ELSIF SpeedUpSubState=SpeedUpCS AND gait_cycle-EnterSpeedUpCSCount=LREAL_TO_UDINT(Time_CS*gvl.sampleRate) THEN
	SpeedUpSubState:=SpeedUpDS;
	EnterSpeedUpDSCount:=gait_cycle;
	body_ref_pos_enter :=body_ref_pos;
	body_ref_ang_enter:=body_ref_ang;
	leg_ref_pos_enter := leg_ref_pos;
ELSIF SpeedUpSubState=SpeedUpDS AND gait_cycle-EnterSpeedUpDSCount=LREAL_TO_UDINT(Time_DS*gvl.sampleRate) THEN
	SpeedUpSubState:=SpeedUpSS;
	EnterSpeedUpSPCount:=gait_cycle;
	body_ref_pos_enter :=body_ref_pos;
	body_ref_ang_enter:=body_ref_ang;
	leg_ref_pos_enter := leg_ref_pos;
	SpeedUpFinished:=TRUE;
	tipForceDesire:=tipForceDesireZeros;
	RequireSlide:=TRUE;
END_IF

body_ref_pos:=body_ref_pos_enter;
body_ref_ang:=body_ref_ang_enter;
leg_ref_pos:=leg_ref_pos_enter;

IF SpeedUpSubState=SpeedUpAS AND gait_cycle-EnterSpeedUpASCount<=Time_AS*gvl.sampleRate THEN
	fbHermitInterpolation(t0:=EnterSpeedUpASCount*delta_t , T:=Time_AS , y0:=0 , 
		y1:=Distance_x_AS , v0:=0 , v1:=target_vel , tNow:=gait_cycle* delta_t, 
		y=> body_ref_pos_wrt_body.data[0], v=>invalid );	
	body_ref_pos_wrt_body.data[1]:=0;body_ref_pos_wrt_body.data[2]:=0;
	fbRotMat(yaw := body_ref_ang_enter.data[2], pitch := body_ref_ang_enter.data[1],roll := body_ref_ang_enter.data[0], rm =>  Rb_target1 );
	body_ref_pos:=VecAdd(body_ref_pos_enter,MatMulVec(Rb_target1,body_ref_pos_wrt_body));
	
	//force compensator
	tipForceTarget:=tipForceDesireLegAF;
	IF (gait_cycle-EnterSpeedUpASCount)<=fceLoadTime*gvl.sampleRate THEN
		tr  := UDINT_TO_LREAL(gait_cycle-EnterSpeedUpASCount) / gvl.sampleRate / fceLoadTime;
		fbGetPivot(tNow := tr, tTotal := 1.0, pivot => pvt);
		FOR i:=0 TO 5 DO
			FOR j:=0 TO 2 DO
				tipForceDesire[i,j]:=(1-pvt)*tipForceDesireZeros[i,j]+pvt*tipForceTarget[i,j];
			END_FOR
		END_FOR	
	END_IF
	
END_IF
	//force compensator
	tipForceTarget:=tipForceDesireLegAF;
	IF (gait_cycle-EnterSpeedUpASCount)>(Time_AS+Time_CS-fceLoadTime)*gvl.sampleRate AND (gait_cycle-EnterSpeedUpASCount)<=(Time_AS+Time_CS)*gvl.sampleRate THEN
		tr  := (UDINT_TO_LREAL(gait_cycle-EnterSpeedUpASCount) / gvl.sampleRate- (Time_AS+Time_CS-fceLoadTime))/ fceLoadTime;
		fbGetPivot(tNow := tr, tTotal := 1.0, pivot => pvt);
		FOR i:=0 TO 5 DO
			FOR j:=0 TO 2 DO
				tipForceDesire[i,j]:=(1-pvt)*tipForceTarget[i,j]+pvt*tipForceDesireZeros[i,j];
			END_FOR
		END_FOR	
	END_IF

IF SpeedUpSubState=SpeedUpCS AND gait_cycle-EnterSpeedUpCSCount<=Time_CS*gvl.sampleRate THEN
	fbHermitInterpolation(t0:=EnterSpeedUpCSCount*delta_t , T:=Time_CS , y0:=0 , 
		y1:=target_vel*Time_CS , v0:=target_vel , v1:=target_vel , tNow:=gait_cycle* delta_t, 
		y=> body_ref_pos_wrt_body.data[0], v=>invalid );
	body_ref_pos_wrt_body.data[1]:=0;body_ref_pos_wrt_body.data[2]:=0;
	fbRotMat(yaw := body_ref_ang_enter.data[2], pitch := body_ref_ang_enter.data[1],roll := body_ref_ang_enter.data[0], rm =>  Rb_target1 );
	body_ref_pos:=VecAdd(body_ref_pos_enter,MatMulVec(Rb_target1,body_ref_pos_wrt_body));
END_IF
IF SpeedUpSubState=SpeedUpDS AND gait_cycle-EnterSpeedUpDSCount<=Time_DS*gvl.sampleRate THEN
	fbHermitInterpolation(t0:=EnterSpeedUpDSCount*delta_t , T:=Time_DS , y0:=0 , 
		y1:=Distance_x_DS , v0:=target_vel , v1:=0 , tNow:=gait_cycle* delta_t, 
		y=> body_ref_pos_wrt_body.data[0], v=>invalid );
	body_ref_pos_wrt_body.data[1]:=0;body_ref_pos_wrt_body.data[2]:=0;
	
	fbRotMat(yaw := body_ref_ang_enter.data[2], pitch := body_ref_ang_enter.data[1],roll := body_ref_ang_enter.data[0], rm =>  Rb_target1 );
	body_ref_pos:=VecAdd(body_ref_pos_enter,MatMulVec(Rb_target1,body_ref_pos_wrt_body));
	
	tr  := UDINT_TO_LREAL(gait_cycle - EnterSpeedUpDSCount) / gvl.sampleRate / Time_DS;
	fbGetPivot(tNow := tr, tTotal := 1.0, pivot => pvt);
	FOR i:=0 TO 1 DO
		leg_ref_pos[Mapping05[i]].data[2]:=(1-pvt)*leg_ref_pos_enter[Mapping05[i]].data[2]+pvt*(leg_ref_pos_enter[Mapping05[i]].data[2]+Distance_y_DS);
	END_FOR
	
END_IF
IF SpeedUpSubState=SpeedUpAS OR SpeedUpSubState=SpeedUpCS OR SpeedUpSubState=SpeedUpDS THEN
	FOR i:=0 TO 1 DO
		gvl.legCtrl[Mapping14[i]].ForwardKinetics(motorAngles:=SpeedUp_MJntRef[i].data , legIndex:=Mapping14[i] , tipPosition=>SpeedUp_MPosWrtHip[i].data );
		gvl.legCtrl[Mapping23[i]].ForwardKinetics(motorAngles:=SpeedUp_FJntRef[i].data , legIndex:=Mapping23[i] , tipPosition=>SpeedUp_FPosWrtHip[i].data );
		fbRotMat(yaw := body_ref_ang_enter.data[2], pitch := body_ref_ang_enter.data[1],roll := body_ref_ang_enter.data[0], rm =>  Rb_target1 );
		temp.data[0]:=hip_pos[Mapping14[i],0];temp.data[1]:=hip_pos[Mapping14[i],1];temp.data[2]:=hip_pos[Mapping14[i],2];
		leg_ref_pos[Mapping14[i]]:= VecAdd( MatMulVec(Rb_target1, VecAdd(temp,MatMulVec(Rleg[Mapping14[i]],SpeedUp_MPosWrtHip[i]))),body_ref_pos);
		temp.data[0]:=hip_pos[Mapping23[i],0];temp.data[1]:=hip_pos[Mapping23[i],1];temp.data[2]:=hip_pos[Mapping23[i],2];
		leg_ref_pos[Mapping23[i]]:= VecAdd( MatMulVec(Rb_target1, VecAdd(temp,MatMulVec(Rleg[Mapping23[i]],SpeedUp_FPosWrtHip[i]))),body_ref_pos);
	END_FOR
END_IF
END_METHOD

METHOD PUBLIC TrjPlanning_StoneRot : BOOL
VAR_INPUT
END_VAR
VAR
	(*StoneRot_FJntTarget:ARRAY[0..1,0..2] OF LREAL:=[-90*pi/180,524*pi/180,-190*pi/180,
                                                     90*pi/180,524*pi/180,-190*pi/180];*)
													 
	(*StoneRot_FJntTarget:ARRAY[0..1,0..2] OF LREAL:=[-90*pi/180,165*pi/180,(-190+360)*pi/180,
                                                     90*pi/180,165*pi/180,(-190+360)*pi/180];	//164 lose,165T 170S lose;*)
	StoneRot_FJntTarget:ARRAY[0..1,0..2] OF LREAL:=[-90*pi/180,167*pi/180,(171)*pi/180,
                                                     90*pi/180,167*pi/180,(171)*pi/180];	//164 lose,166T 168S passive wheels colide;												 
	tr: LREAL;
	i: INT;
	Rb_target1: Mat3;	
	temp:vec3;										 
	j: INT;
	noPlanning: BOOL;
END_VAR
//*****************************test trajectory*****************************************

	FOR i:=0 TO 1 DO
		(*IF SetColide=TRUE THEN
			gvl.tipActualFce[Mapping23[i],2]:=100;
		END_IF	*)
		(*IF(gait_cycle-EnterStoneRotCount)=0.5*StoneGripTime*gvl.sampleRate THEN
			gvl.tipActualFce[Mapping23[i],2]:=100;
		END_IF *)
		noPlanning:=TRUE;
	END_FOR
	

//**********************************end************************************************	

(*FOR i:=0 TO 1 DO
	IF StoneRotSubState[i]=FALSE AND isStone(Mapping23[i]) THEN
		StoneRotSubState[i]:=TRUE;
		leg_ref_pos_enter[Mapping23[i]]:=leg_ref_pos[Mapping23[i]];
	END_IF
END_FOR*)

IF (StoneRotSubState[0]=FALSE OR StoneRotSubState[1]=FALSE) AND (gait_cycle-EnterStoneRotCount)=LREAL_TO_UDINT(StoneGripTime*gvl.sampleRate) THEN
	StoneRotSubState[0]:=TRUE;
	StoneRotSubState[1]:=TRUE;
	leg_ref_pos_enter[Mapping23[0]]:=leg_ref_pos[Mapping23[0]];
	leg_ref_pos_enter[Mapping23[1]]:=leg_ref_pos[Mapping23[1]];
END_IF
	
body_ref_pos:=body_ref_pos_enter;
body_ref_ang:=body_ref_ang_enter;
leg_ref_pos:=leg_ref_pos_enter;


	IF (gait_cycle-EnterStoneRotCount)<=StoneGripTime*gvl.sampleRate THEN
		FOR i:=0 TO 1 DO
			IF StoneRotSubState[i]=FALSE THEN
			tr  := UDINT_TO_LREAL(gait_cycle - EnterStoneRotCount) / gvl.sampleRate /StoneGripTime;
			fbGetPivot(tNow := tr, tTotal := 1.0, pivot => pvt);
			FOR j:=0 TO 2 DO
				StoneRot_FJntRef[i].data[j]:=(1-pvt)*StoneRot_FJntStart[i].data[j]+pvt*(StoneRot_FJntTarget[i,j]);
			END_FOR
			gvl.legCtrl[Mapping23[i]].ForwardKinetics(motorAngles:=StoneRot_FJntRef[i].data , legIndex:=Mapping23[i] , tipPosition=>StoneRot_FPosWrtHip[i].data );
			fbRotMat(yaw := body_ref_ang_enter.data[2], pitch := body_ref_ang_enter.data[1],roll := body_ref_ang_enter.data[0], rm =>  Rb_target1 );
			temp.data[0]:=hip_pos[Mapping23[i],0];temp.data[1]:=hip_pos[Mapping23[i],1];temp.data[2]:=hip_pos[Mapping23[i],2];
			leg_ref_pos[Mapping23[i]]:= VecAdd( MatMulVec(Rb_target1, VecAdd(temp,MatMulVec(Rleg[Mapping23[i]],StoneRot_FPosWrtHip[i]))),body_ref_pos);
			END_IF
		END_FOR
	ELSE
		noPlanning:=TRUE;
	END_IF

IF (gait_cycle-EnterStoneRotCount)>StoneGripTime*gvl.sampleRate  THEN
		stone_rot_vel:=GVL.stone_rot_vel/60*2*pi;
		GVL.jogVelocity[18]:=stone_rot_vel;
		GVL.jogVelocity[19]:=-stone_rot_vel;
		FOR j:=18 TO 19 DO
			gvl.motorDrive[j].SetTrgVel(GVL.jogVelocity[j]);
			IF gvl.motorDrive[j].cvSetVel = GVL.jogVelocity[j] THEN
				gvl.jogButton[j]:=FALSE;
			ELSE
				gvl.jogButton[j]:=TRUE;
			END_IF
		END_FOR
END_IF

IF StoneRotFinished=FALSE AND (gait_cycle-EnterStoneRotCount)>=(StoneGripTime+StoneRotTime)*gvl.sampleRate THEN
	StoneRotFinished:=TRUE;
END_IF
END_METHOD

END_FUNCTION_BLOCK

// ---- POUs/GaitPlanner/RcToCurlingFromSlip.TcPOU
FUNCTION_BLOCK RcToCurlingFromSlip
VAR_INPUT
END_VAR
VAR_OUTPUT
END_VAR
VAR
//*********************************common state start*********************************************	
	gait_cycle : UDINT := 0;
	quit_flag : BOOL := FALSE;
	delta_t:LREAL:=0.001;//sampling period
	isFinished:BOOL:=FALSE;
	// robot geometrical parameters
	hip_pos : ARRAY[0..5, 0..2] OF LREAL := [-0.369,  -0.125, 0,
                                             0,  -0.28, 0,
                                             0.36, -0.125, 0,
                                             0.36, 0.125, 0,
											 0,0.28,0,
											 -0.369,0.125,0];

	leg_index_mapping : ARRAY[0..5] OF INT := [1, 2, 3, 4,5,6];
	Rleg : ARRAY[0..5] OF Mat3;
	
	joint_ref_pos_init : ARRAY[0..5] OF Vec3;
	jointPosLast   : ARRAY[0..5, 0..2] OF LREAL; 
	
	body_ref_pos_init : Vec3;
	body_ref_ang_init : Vec3;
    leg_ref_pos_init : ARRAY[0..5] OF Vec3;
	leg_ref_pos_init_wrt_hip : ARRAY[0..5] OF Vec3;
	
	body_ref_pos_enter : Vec3;
	body_ref_ang_enter : Vec3;
    leg_ref_pos_enter : ARRAY[0..5] OF Vec3;
	
	body_ref_pos : Vec3;
	body_ref_ang : Vec3;
    leg_ref_pos : ARRAY[0..5] OF Vec3;
	leg_ref_pos_wrt_hip : ARRAY[0..5] OF Vec3;
	
	body_ref_pos_next : Vec3;
	body_ref_ang_next : Vec3;
    leg_ref_pos_next : ARRAY[0..5] OF Vec3;
	leg_ref_pos_next_wrt_hip : ARRAY[0..5] OF Vec3;
	leg_ref_vel_next_wrt_hip : ARRAY[0..5] OF Vec3;
	
	// output test
	joint_ref_pos   : ARRAY[0..5] OF Vec3;
	joint_ref_vel   : ARRAY[0..5] OF Vec3;
	
	jointPosTarget  : ARRAY[0..5, 0..2] OF LREAL; 
	jointVelTarget  : ARRAY[0..5, 0..2] OF LREAL;  
	jointFceTarget  : ARRAY[0..5, 0..2] OF LREAL;  
	
	pvt, pvtDot : LREAL;
	
	fbRotmat : RotM;
	fbGetPivot  : GetPivot;
	fbCubicSpline:CubicSpline;
	
	Mapping05:ARRAY[0..1] OF INT:=[0,5];
	Mapping14:ARRAY[0..1] OF INT:=[1,4];
	Mapping23:ARRAY[0..1] OF INT:=[2,3];
//*********************************common state end*********************************************

//*********************************exclusive state start****************************************
	BJntStart:ARRAY[0..1] OF vec3;
	BPosWrtHip:ARRAY[0..1] OF vec3;
	BJntRef:ARRAY[0..1] OF vec3;
	
	BJntRetract:ARRAY[0..1,0..2] OF LREAL;
	BJntExtend:ARRAY[0..1,0..2] OF LREAL;	
	BlegCenterType:UINT:=0;//0 is double pedals, 1 is single pedals
	BPosExtendRefDouble:ARRAY[0..1,0..2] OF LREAL:=[-0.15,-0.1687,0,
                                                     -0.15,-0.1687,0];
	BPosExtendRefSingle:ARRAY[0..1,0..2] OF LREAL:=[-0.15,-0.1687,-0.05,
                                                     -0.15,-0.1687,0.05];	
	BPosExtractRef:ARRAY[0..1,0..2]      OF LREAL:=[-0.15,-0.1687+0.08,-0.05,
                                                     -0.15,-0.1687+0.08,0.05];
												 
	BJntRetractRef:ARRAY[0..1,0..2] OF LREAL:=[0*pi/180,130.6330*pi/180,290.5615*pi/180,
                                            0*pi/180,130.6330*pi/180,290.5615*pi/180];
								   

	FJntStart:ARRAY[0..1] OF vec3;
	FPosWrtHip:ARRAY[0..1] OF vec3;
	FJntRef:ARRAY[0..1] OF vec3;	
	FJntGrip:ARRAY[0..1,0..2] OF LREAL:=[-90*pi/180,(522-360)*pi/180,(-188+360)*pi/180,
                                        90*pi/180,(522-360)*pi/180,(-188+360)*pi/180];		
	MJntStart:ARRAY[0..1] OF vec3;
	MPosWrtHip:ARRAY[0..1] OF vec3;
	MJntRef:ARRAY[0..1] OF vec3;	
	MJntLiftTarget:ARRAY[0..1,0..2] OF LREAL;
	MPosLiftTarget:ARRAY[0..1,0..2] OF LREAL:=[-0.0141,-0.1797+0.05,-0.1246,
                                               -0.0141,-0.1797+0.05,0.1246];	
	MJntLiftTargetRef:ARRAY[0..1,0..2] OF LREAL:=[0,331.45*pi/180,-149*pi/180,
                                               0,331.45*pi/180,-149*pi/180];	
	BRetractTime:LREAL:=2;
	BExtendTime:LREAL:=2;
	FGripTime:LREAL:=2;		
	MLiftTime:LREAL:=2;	
	
	isBMove: BOOL:=FALSE;	
	isMMove: BOOL:=FALSE;	
	isFMove: BOOL:=FALSE;	
	enterMMoveCount:UDINT;	
	enterFMoveCount:UDINT;			
//*********************************exclusive state end****************************************
END_VAR

METHOD PUBLIC DoPlanning : BOOL
VAR_INPUT
	count : UDINT;
END_VAR
VAR
	i, j  : INT;
	tempLeg:ARRAY [0..2] OF LREAL;
	tempJnt:ARRAY [0..2] OF LREAL;
	tempRef:ARRAY [0..2] OF LREAL;
END_VAR
IF count = 0 THEN
	isFinished := FALSE;
	Initialize();
	IF BlegCenterType=0 THEN
		FOR i:=0 TO 1 DO
			tempLeg[0]:=BPosExtendRefDouble[i,0];tempLeg[1]:=BPosExtendRefDouble[i,1];tempLeg[2]:=BPosExtendRefDouble[i,2];
			tempRef[0]:=BJntRetractRef[i,0];tempRef[1]:=BJntRetractRef[i,1];tempRef[2]:=BJntRetractRef[i,2];
			GVL.legCtrl[Mapping05[i]].InverseKinetics(tipPosition:=tempLeg , refPosLast:=tempRef , legIndex:=Mapping05[i] , motorAngles=>tempJnt , isSingular=> );
			BJntExtend[i,0]:=tempJnt[0];BJntExtend[i,1]:=tempJnt[1];BJntExtend[i,2]:=tempJnt[2];
		END_FOR		
	ELSE
		FOR i:=0 TO 1 DO
			tempLeg[0]:=BPosExtendRefSingle[i,0];tempLeg[1]:=BPosExtendRefSingle[i,1];tempLeg[2]:=BPosExtendRefSingle[i,2];
			tempRef[0]:=BJntRetractRef[i,0];tempRef[1]:=BJntRetractRef[i,1];tempRef[2]:=BJntRetractRef[i,2];
			GVL.legCtrl[Mapping05[i]].InverseKinetics(tipPosition:=tempLeg , refPosLast:=tempRef , legIndex:=Mapping05[i] , motorAngles=>tempJnt , isSingular=> );
			BJntExtend[i,0]:=tempJnt[0];BJntExtend[i,1]:=tempJnt[1];BJntExtend[i,2]:=tempJnt[2];	
		END_FOR		
	END_IF
	FOR i:=0 TO 1 DO
		tempLeg[0]:=BPosExtractRef[i,0];tempLeg[1]:=BPosExtractRef[i,1];tempLeg[2]:=BPosExtractRef[i,2];
		tempRef[0]:=BJntRetractRef[i,0];tempRef[1]:=BJntRetractRef[i,1];tempRef[2]:=BJntRetractRef[i,2];
		GVL.legCtrl[Mapping05[i]].InverseKinetics(tipPosition:=tempLeg , refPosLast:=tempRef , legIndex:=Mapping05[i] , motorAngles=>tempJnt , isSingular=> );
		BJntRetract[i,0]:=tempJnt[0];BJntRetract[i,1]:=tempJnt[1];BJntRetract[i,2]:=tempJnt[2];
	END_FOR

	FOR i:=0 TO 1 DO
		tempLeg[0]:=MPosLiftTarget[i,0];tempLeg[1]:=MPosLiftTarget[i,1];tempLeg[2]:=MPosLiftTarget[i,2];
		tempRef[0]:=MJntLiftTargetRef[i,0];tempRef[1]:=MJntLiftTargetRef[i,1];tempRef[2]:=MJntLiftTargetRef[i,2];
		GVL.legCtrl[Mapping14[i]].InverseKinetics(tipPosition:=tempLeg , refPosLast:=tempRef , legIndex:=Mapping14[i] , motorAngles=>tempJnt , isSingular=> );
		MJntLiftTarget[i,0]:=tempJnt[0];MJntLiftTarget[i,1]:=tempJnt[1];MJntLiftTarget[i,2]:=tempJnt[2];
	END_FOR		
	
END_IF

TrjPlanning();

IF quit_flag THEN
	isFinished := TRUE;
	quit_flag := FALSE;
END_IF
END_METHOD

METHOD PUBLIC Initialize : BOOL
VAR_INPUT
END_VAR
VAR
	i, j : INT;
	sum_height : LREAL := 0;
	leg_pos    : ARRAY[0..2] OF LREAL;
	
	Rb : Mat3;
	hip_pos_j  : Vec3;
	leg_pos_wrt_com : Vec3;
	
END_VAR
Rleg[0]:=SetMat3(1,0,0,0,0,-1,0,1,0);
Rleg[1]:=SetMat3(-1,0,0,0,0,1,0,1,0,);
Rleg[2]:=SetMat3(-1,0,0,0,0,1,0,1,0);
Rleg[3]:=SetMat3(-1,0,0,0,0,1,0,1,0);
Rleg[4]:=SetMat3( -1,0,0,0,0,1,0,1,0);
Rleg[5]:=SetMat3(1,0,0,0,0,-1,0,1,0);

quit_flag  := FALSE;
gait_cycle := 0;
isBMove:=TRUE;
isMMove:=FALSE;
delta_t:=1.0/gvl.sampleRate;

FOR i := 0 TO 5 DO
	FOR j := 0 TO 2 DO
		IF ABS(gvl.jntLastRefPos[i, j] - gvl.jntActualPos[i, j]) < 0.2 THEN
			joint_ref_pos_init[i].data[j] := gvl.jntLastRefPos[i, j];
		ELSE
			joint_ref_pos_init[i].data[j] := gvl.jntActualPos[i, j];
		END_IF
		jointPosLast[i,j]:=joint_ref_pos_init[i].data[j];
	END_FOR
END_FOR

sum_height := 0;
FOR j := 0 TO 5 DO
	// FK
	gvl.legCtrl[j].ForwardKinetics(motorAngles := joint_ref_pos_init[j].data, legIndex:=j, tipPosition => leg_pos);
	leg_ref_pos_init_wrt_hip[j] := SetVec3(leg_pos[0], leg_pos[1], leg_pos[2]);
	sum_height := sum_height - leg_ref_pos_init_wrt_hip[j].data[1];
END_FOR
body_ref_pos_init := SetVec3(0, 0, sum_height/6.0);
body_ref_ang_init := SetVec3(0, 0, 0);                            

FOR j := 0 TO 5 DO
	fbRotMat(yaw := body_ref_ang_init.data[2],
             pitch := body_ref_ang_init.data[1],
             roll := body_ref_ang_init.data[0],
             rm => Rb );
	hip_pos_j := SetVec3(hip_pos[j, 0], hip_pos[j, 1], hip_pos[j, 2]);
	leg_pos_wrt_com := VecAdd(MatMulVec(Rleg[j], leg_ref_pos_init_wrt_hip[j]), hip_pos_j);
    leg_ref_pos_init[j] := VecAdd(body_ref_pos_init, MatMulVec(Rb, leg_pos_wrt_com));
END_FOR

body_ref_pos := body_ref_pos_init;
body_ref_ang := body_ref_ang_init;
leg_ref_pos := leg_ref_pos_init;
leg_ref_pos_wrt_hip := leg_ref_pos_init_wrt_hip;

body_ref_pos_enter := body_ref_pos_init;
body_ref_ang_enter := body_ref_ang_init;
leg_ref_pos_enter := leg_ref_pos_init;

FOR i:=0 TO 1 DO
	FOR j:=0 TO 2 DO
		BJntStart[i].data[j]:=joint_ref_pos_init[Mapping05[i]].data[j];
		MJntStart[i].data[j]:=joint_ref_pos_init[Mapping14[i]].data[j];
		FJntStart[i].data[j]:=joint_ref_pos_init[Mapping23[i]].data[j];
	END_FOR
END_FOR

FOR i := 0 TO 5 DO
	FOR j := 0 TO 2 DO
		jointPosTarget[i, j] := joint_ref_pos_init[i].data[j];
		jointVelTarget[i, j] := 0;
		jointFceTarget[i, j] := 0;
	END_FOR
END_FOR
END_METHOD

METHOD PUBLIC TrjPlanning : BOOL
VAR_INPUT
END_VAR

VAR
	tr: lreal;
	i: INT;
	j: INT;
	Rb_target1: Mat3;
	temp: vec3;
	
	Rb: Mat3;
	hip_pos_j: Vec3;
	leg_ref_pos_wrt_com_j: Vec3;
	tmp: Vec3;
	tip_pos: Vec3;
	tip_vel: Vec3;
	jointTmpPosLast: ARRAY [0..2] OF LREAL;
END_VAR
gait_cycle := gait_cycle + 1;

IF gait_cycle=(BRetractTime+BExtendTime)*gvl.sampleRate OR (gait_cycle-enterMMoveCount) =MLiftTime*gvl.sampleRate OR (gait_cycle-enterFMoveCount)=FGripTime*gvl.sampleRate THEN
	leg_ref_pos_enter:=leg_ref_pos;
END_IF

IF isMMove=FALSE AND isFMove=FALSE THEN
IF isBMove=TRUE THEN
	body_ref_pos:=body_ref_pos_enter;
	body_ref_ang:=body_ref_ang_enter;
	leg_ref_pos:=leg_ref_pos_enter;
	IF gait_cycle<=BRetractTime*gvl.sampleRate  THEN
		tr  := UDINT_TO_LREAL(gait_cycle) / gvl.sampleRate /BRetractTime;
		fbGetPivot(tNow := tr, tTotal := 1.0, pivot => pvt);
		FOR i:=0 TO 1 DO
			FOR j:=0 TO 2 DO
				BJntRef[i].data[j]:=(1-pvt)*BJntStart[i].data[j]+pvt*(BJntRetract[i,j]);
			END_FOR
			gvl.legCtrl[Mapping05[i]].ForwardKinetics(motorAngles:=BJntRef[i].data , legIndex:=Mapping05[i] , tipPosition=>BPosWrtHip[i].data );
			fbRotMat(yaw := body_ref_ang_init.data[2], pitch := body_ref_ang_init.data[1],roll := body_ref_ang_init.data[0], rm =>  Rb_target1 );
			temp.data[0]:=hip_pos[Mapping05[i],0];temp.data[1]:=hip_pos[Mapping05[i],1];temp.data[2]:=hip_pos[Mapping05[i],2];
			leg_ref_pos[Mapping05[i]]:= VecAdd( MatMulVec(Rb_target1, VecAdd(temp,MatMulVec(Rleg[Mapping05[i]],BPosWrtHip[i]))),body_ref_pos);
		END_FOR
	ELSIF gait_cycle<=(BRetractTime+BExtendTime)*gvl.sampleRate THEN
		tr  := (UDINT_TO_LREAL(gait_cycle) / gvl.sampleRate- BRetractTime)/BExtendTime;
		fbGetPivot(tNow := tr, tTotal := 1.0, pivot => pvt);
		FOR i:=0 TO 1 DO
			FOR j:=0 TO 2 DO
				BJntRef[i].data[j]:=(1-pvt)*BJntRetract[i,j]+pvt*BJntExtend[i,j];
			END_FOR
			gvl.legCtrl[Mapping05[i]].ForwardKinetics(motorAngles:=BJntRef[i].data , legIndex:=Mapping05[i] , tipPosition=>BPosWrtHip[i].data );
			fbRotMat(yaw := body_ref_ang_init.data[2], pitch := body_ref_ang_init.data[1],roll := body_ref_ang_init.data[0], rm =>  Rb_target1 );
			temp.data[0]:=hip_pos[Mapping05[i],0];temp.data[1]:=hip_pos[Mapping05[i],1];temp.data[2]:=hip_pos[Mapping05[i],2];
			leg_ref_pos[Mapping05[i]]:= VecAdd( MatMulVec(Rb_target1, VecAdd(temp,MatMulVec(Rleg[Mapping05[i]],BPosWrtHip[i]))),body_ref_pos);
		END_FOR
	ELSE
		isBMove:=FALSE;
		isMMove:=TRUE;
		//leg_ref_pos_enter:=leg_ref_pos;
		enterMMoveCount:=gait_cycle;
	END_IF
END_IF
END_IF

IF isBMove=FALSE AND isFMove=FALSE THEN
IF isMMove=TRUE THEN
	body_ref_pos:=body_ref_pos_enter;
	body_ref_ang:=body_ref_ang_enter;
	leg_ref_pos:=leg_ref_pos_enter;
	IF (gait_cycle-enterMMoveCount) <=MLiftTime*gvl.sampleRate THEN
		tr  := UDINT_TO_LREAL(gait_cycle- enterMMoveCount) / gvl.sampleRate/MLiftTime;
		fbGetPivot(tNow := tr, tTotal := 1.0, pivot => pvt);
		FOR i:=0 TO 1 DO
			FOR j:=0 TO 2 DO	
				MJntRef[i].data[j]:=(1-pvt)*MJntStart[i].data[j]+pvt*(MJntLiftTarget[i,j]);
			END_FOR
			gvl.legCtrl[Mapping14[i]].ForwardKinetics(motorAngles:=MJntRef[i].data , legIndex:=Mapping14[i] , tipPosition=>MPosWrtHip[i].data );
			fbRotMat(yaw := body_ref_ang_init.data[2], pitch := body_ref_ang_init.data[1],roll := body_ref_ang_init.data[0], rm =>  Rb_target1 );
			temp.data[0]:=hip_pos[Mapping14[i],0];temp.data[1]:=hip_pos[Mapping14[i],1];temp.data[2]:=hip_pos[Mapping14[i],2];
			leg_ref_pos[Mapping14[i]]:= VecAdd( MatMulVec(Rb_target1, VecAdd(temp,MatMulVec(Rleg[Mapping14[i]],MPosWrtHip[i]))),body_ref_pos);
		END_FOR
	ELSE
		isMMove:=FALSE;
		isFMove:=TRUE;
		//leg_ref_pos_enter:=leg_ref_pos;
		enterFMoveCount:=gait_cycle;
	END_IF
END_IF
END_IF

IF isBMove=FALSE AND isMMove=FALSE THEN
IF isFMove=TRUE THEN
	body_ref_pos:=body_ref_pos_enter;
	body_ref_ang:=body_ref_ang_enter;
	leg_ref_pos:=leg_ref_pos_enter;
	IF (gait_cycle-enterFMoveCount) <=FGripTime*gvl.sampleRate THEN
		tr  := UDINT_TO_LREAL(gait_cycle- enterFMoveCount) / gvl.sampleRate/FGripTime;
		fbGetPivot(tNow := tr, tTotal := 1.0, pivot => pvt);
		FOR i:=0 TO 1 DO
			FOR j:=0 TO 2 DO	
				FJntRef[i].data[j]:=(1-pvt)*FJntStart[i].data[j]+pvt*(FJntGrip[i,j]);
			END_FOR
		gvl.legCtrl[Mapping23[i]].ForwardKinetics(motorAngles:=FJntRef[i].data , legIndex:=Mapping23[i] , tipPosition=>FPosWrtHip[i].data );
		fbRotMat(yaw := body_ref_ang_init.data[2], pitch := body_ref_ang_init.data[1],roll := body_ref_ang_init.data[0], rm =>  Rb_target1 );
		temp.data[0]:=hip_pos[Mapping23[i],0];temp.data[1]:=hip_pos[Mapping23[i],1];temp.data[2]:=hip_pos[Mapping23[i],2];
		leg_ref_pos[Mapping23[i]]:= VecAdd( MatMulVec(Rb_target1, VecAdd(temp,MatMulVec(Rleg[Mapping23[i]],FPosWrtHip[i]))),body_ref_pos);
		END_FOR
	ELSE
		isFMove:=FALSE;
		isFinished := TRUE;
		//leg_ref_pos_enter:=leg_ref_pos;
	END_IF
END_IF
END_IF

// transform TO leg local frame AND DO inverse kinematics
FOR j := 0 TO 5 DO
	fbRotMat(
    	yaw := body_ref_ang.data[2], 
		pitch := body_ref_ang.data[1], 
		roll := body_ref_ang.data[0], 
		rm => Rb);
	hip_pos_j := SetVec3(hip_pos[j, 0], hip_pos[j, 1], hip_pos[j, 2]);

	//leg_ref_pos_wrt_com = Rb' * (leg_ref_pos - body_ref_pos)
	leg_ref_pos_wrt_com_j := MatMulVec(
		                         MatTranspose(Rb),
								 VecAdd(
									 leg_ref_pos[j],
									 VecNeg(body_ref_pos)
                                 )
                             );
	// leg_ref_pos_wrt_hip = Rleg' * (leg_ref_pos_wrt_com_j - hip_pos)
	leg_ref_pos_next_wrt_hip[j] := MatMulVec(
		                               MatTranspose(Rleg[j]),
									   VecAdd(
										   leg_ref_pos_wrt_com_j,
										   VecNeg(hip_pos_j)
									   )
								   );
								   
	leg_ref_vel_next_wrt_hip[j] := VecMulNum(VecAdd(leg_ref_pos_next_wrt_hip[j], VecNeg(leg_ref_pos_wrt_hip[j])), DINT_TO_LREAL(gvl.sampleRate));
END_FOR


// mapping to actual joints
FOR j := 0 TO 5 DO
	tmp := leg_ref_pos_next_wrt_hip[leg_index_mapping[j]-1];
	tip_pos := SetVec3(tmp.data[0], tmp.data[1], tmp.data[2]);
	tmp := leg_ref_vel_next_wrt_hip[leg_index_mapping[j]-1];
	tip_vel := SetVec3(tmp.data[0], tmp.data[1], tmp.data[2]);
	FOR i:= 0 TO 2 DO
		jointTmpPosLast[i]:=jointPosLast[j,i];
	END_FOR		
	gvl.legCtrl[j].InversePosAndVel(
		tipPos := tip_pos.data, 
		tipVel := tip_vel.data, 
		refPosLast:=jointTmpPosLast,
		legIndex:=j,
		jntPos => joint_ref_pos[j].data, 
		jntVel => joint_ref_vel[j].data);
	
END_FOR

// link to physical outputs
FOR i := 0 TO 5 DO
	FOR j := 0 TO 2 DO
		jointPosTarget[i, j] := joint_ref_pos[i].data[j];
		jointPosLast[i,j]:=jointPosTarget[i, j] ;
		jointVelTarget[i, j] := joint_ref_vel[i].data[j];
		jointFceTarget[i, j] := 0;
	END_FOR
END_FOR

// store refs for next loop
leg_ref_pos_wrt_hip := leg_ref_pos_next_wrt_hip;
END_METHOD

END_FUNCTION_BLOCK

// ---- POUs/GaitPlanner/RcToStanceFromSlip.TcPOU
FUNCTION_BLOCK RcToStanceFromSlip
VAR_INPUT
END_VAR
VAR_OUTPUT
END_VAR
VAR
	tTotalAll     : LREAL := 5000;
	
	// robot geometrical parameters
	hip_pos : ARRAY[0..5, 0..2] OF LREAL := [-0.369,  -0.125, 0,
                                             0,  -0.28, 0,
                                             0.36, -0.125, 0,
                                             0.36, 0.125, 0,
											 0,0.28,0,
											 -0.369,0.125,0];

	leg_index_mapping : ARRAY[0..5] OF INT := [1, 2, 3, 4,5,6];
	Rleg : ARRAY[0..5] OF Mat3;
	
	gait_cycle : UDINT := 0;
	quit_flag : BOOL := FALSE;
	
	joint_ref_pos_init : ARRAY[0..5] OF Vec3;
	jointPosLast   : ARRAY[0..5, 0..2] OF LREAL; 
	
	body_ref_pos_init : Vec3;
	body_ref_ang_init : Vec3;
    leg_ref_pos_init : ARRAY[0..5] OF Vec3;
	leg_ref_pos_init_wrt_hip : ARRAY[0..5] OF Vec3;

	body_ref_pos : Vec3;
	body_ref_ang : Vec3;
	body_ref_angvel:vec3;
    leg_ref_pos : ARRAY[0..5] OF Vec3;
	leg_ref_pos_wrt_hip : ARRAY[0..5] OF Vec3;
	body_ref_pos_enter : Vec3;
	body_ref_ang_enter : Vec3;
    leg_ref_pos_enter : ARRAY[0..5] OF Vec3;
	leg_ref_pos_wrt_hip_enter : ARRAY[0..5] OF Vec3;
	
	body_ref_pos_next : Vec3;
	body_ref_ang_next : Vec3;
    leg_ref_pos_next : ARRAY[0..5] OF Vec3;
	leg_ref_pos_next_wrt_hip : ARRAY[0..5] OF Vec3;
	leg_ref_vel_next_wrt_hip : ARRAY[0..5] OF Vec3;
	
	// output test
	joint_ref_pos   : ARRAY[0..5] OF Vec3;
	joint_ref_vel   : ARRAY[0..5] OF Vec3;
	
	jointPosTarget  : ARRAY[0..5, 0..2] OF LREAL; 
	jointVelTarget  : ARRAY[0..5, 0..2] OF LREAL;  
	jointFceTarget  : ARRAY[0..5, 0..2] OF LREAL;  
	
	pvt, pvtDot : LREAL;
	
	fbRotmat : RotM;
	fbGetPivot  : GetPivot;
	delta_t:LREAL :=0.0025;//sample time
	
	isFinished : BOOL := FALSE;
	
	//target value from visual system
	adjust_angle_rad:LREAL:=0;//unit:rad
	adjust_angle_actual_rad:LREAL:=0;//unit:rad
	target_vel:LREAL:=0;//unit:m/s
	stone_rot_vel:LREAL:=0;//unit:rad/s
	
	//common variable
	sum_height : LREAL := 0;
	fbElipseInterpolation:ElipseInterpolation;
	fbHermitInterpolation:HermitInterpolation;
	Mapping14:ARRAY[0..1] OF INT:=[1,4];
	Mapping05:ARRAY[0..1] OF INT:=[0,5];
	Mapping23:ARRAY[0..1] OF INT:=[2,3];
	body_target_pos: Vec3;
	
	//state machine 
	state:UINT;
	Ready:UINT:=1;//init state
	BlegCenter:UINT:=2; 
	MlegRollA:UINT:=3;
	FlegRotA:UINT:=4;
	ReduceHeight:UINT:=5;
	MlegRollB:UINT:=6;
	StoneRot:UINT:=7;
	RoughTuning:UINT:=8;
	FineTuning:UINT:=9;
	LiftMleg:UINT:=10;
	SpeedUp:UINT:=11;
	Slide:UINT:=12;
	PushReleaseBall:UINT:=13;
	SpeedDown:UINT:=14;
	MlegRollC:UINT:=15;
	AddHeight:UINT:=16;
	FlegRotB:UINT:=17;
	CurlingFinished:UINT:=18;
	RecoveryReady:UINT:=18;
	
	//contol button
	RequireMlegRollA:BOOL:=FALSE;
	RequireBlegCenter:BOOL:=FALSE;
	RequireFlegRotA:BOOL:=FALSE;
	RequireReduceHeight:BOOL:=FALSE;	
	RequireMlegRollB:BOOL:=FALSE;	
	RequireStoneRot:BOOL:=FALSE;		
	RequireRoughTuning:BOOL:=FALSE;
	RequireFineTuning:BOOL:=FALSE;
	RequireLiftMleg:BOOL:=FALSE;
	RequireSpeedUp:BOOL:=FALSE;
	RequireSlide:BOOL:=FALSE;
	RequirePushReleaseBall:BOOL:=FALSE;
	RequireSpeedDown:BOOL:=FALSE;
	RequireMlegRollC:BOOL:=FALSE;
	RequireAddHeight:BOOL:=FALSE;
	RequireFlegRotB:BOOL:=FALSE;
	RequireRecoveryReady:BOOL:=FALSE;
	
	IsReady:BOOL:=FALSE;
	IsMlegRollA:BOOL:=FALSE;
	IsBlegCenter:BOOL:=FALSE;
	IsFlegRotA:BOOL:=FALSE;
	IsReduceHeight:BOOL:=FALSE;	
	IsMlegRollB:BOOL:=FALSE;	
	IsStoneRot:BOOL:=FALSE;		
	IsRoughTuning:BOOL:=FALSE;
	IsFineTuning:BOOL:=FALSE;
	IsLiftMleg:BOOL:=FALSE;
	IsSpeedUp:BOOL:=FALSE;
	IsSlide:BOOL:=FALSE;
	IsPushReleaseBall:BOOL:=FALSE;
	IsSpeedDown:BOOL:=FALSE;
	IsMlegRollC:BOOL:=FALSE;
	IsAddHeight:BOOL:=FALSE;
	IsFlegRotB:BOOL:=FALSE;
	IsCurlingFinished:BOOL:=FALSE;
	IsRecoveryReady:BOOL:=FALSE;

	ReadyFinished:bool:=false;
	MlegRollAFinished:BOOL:=FALSE;
	BlegCenterFinished:BOOL:=FALSE;
	FlegRotAFinished:BOOL:=FALSE;
	ReduceHeightFinished:BOOL:=FALSE;
	MlegRollBFinished:BOOL:=FALSE;
	StoneRotFinished:BOOL:=FALSE;
	RoughTuningFinished:BOOL:=FALSE;
	FineTuningFinished:BOOL:=FALSE;
	LiftMlegFinished:BOOL:=FALSE;
	SpeedUpFinished:BOOL:=FALSE;
	SlideFinished:BOOL:=FALSE;
	PushReleaseBallFinished:BOOL:=FALSE;
	SpeedDownFinished:BOOL:=FALSE;
	MlegRollCFinished:BOOL:=FALSE;
	AddHeightFinished:BOOL:=FALSE;
	FlegRotBFinished:BOOL:=FALSE;
	RecoveryReadyFinished:BOOL:=FALSE;
	CurlingGaitFinished: BOOL:=FALSE;
	
	EnterMlegRollACount:UDINT;
	EnterBlegCenterCount:UDINT;
	EnterFlegRotACount:UDINT;
	EnterReduceHeightCount:UDINT;
	EnterMlegRollBCount:UDINT;
	EnterStoneRotCount:UDINT;
	EnterRoughTuningCount:UDINT;
	EnterFineTuningCount:UDINT;
	EnterLiftMlegCount:UDINT;
	EnterSpeedUpCount:UDINT;
	EnterSlideCount:UDINT;
	EnterPushReleaseBallCount:UDINT;
	EnterSpeedDownCount:UDINT;
	EnterMlegRollCCount:UDINT;
	EnterAddHeightCount:UDINT;
	EnterFlegRotBCount:UDINT;
	EnterRecoveryReadyCount:UDINT;
		
	//BlegCenter
	BlegCenter_BJntStart:ARRAY[0..1] OF vec3;
	BlegCenter_BPosWrtHip:ARRAY[0..1] OF vec3;
	BlegCenter_BJntRef:ARRAY[0..1] OF vec3;
	BlegCenterRetractTime:LREAL:=2;
	BlegCenterExtendTime:LREAL:=3;
	IsLeg0Move:BOOL:=FALSE;
	IsLeg5Move:BOOL:=FALSE;
	EnterLeg5MoveCount:UDINT;
	
	//MlegRollA
	MlegRollA_MJntStart:ARRAY[0..1] OF vec3;
	MlegRollA_MPosWrtHip:ARRAY[0..1] OF vec3;
	MlegRollA_MJntRef:ARRAY[0..1] OF vec3;
	MlegRollATime:LREAL:=3;
	
	//FlegRotA
	FlegRotA_FJntStart:ARRAY[0..1] OF vec3;
	FlegRotA_FPosWrtHip:ARRAY[0..1] OF vec3;
	FlegRotA_FJntRef:ARRAY[0..1] OF vec3;
	FlegRotATime:LREAL:=3;
	
	//ReduceHeight
	ReduceHeight_FJntRef:ARRAY[0..1] OF vec3;
	ReduceHeight_FPosWrtHip:ARRAY[0..1] OF vec3;
	ReduceHeightTime:LREAL:=3;
	targetHeight:LREAL:=0.1797;//need be calibrated
	
	//MlegRollB
	MlegRollB_MJntStart:ARRAY[0..1] OF vec3;
	MlegRollB_MPosWrtHip:ARRAY[0..1] OF vec3;
	MlegRollB_MJntRef:ARRAY[0..1] OF vec3;
	MlegRollBTime:LREAL:=3;
	
	//StoneRot
	StoneRot_FJntStart:ARRAY[0..1] OF vec3;
	StoneRot_FPosWrtHip:ARRAY[0..1] OF vec3;
	StoneRot_FJntRef:ARRAY[0..1] OF vec3;
	StoneGripTime:LREAL:=3;
	StoneRotSubState:ARRAY [0..1] OF BOOL:=[FALSE,FALSE];
	StoneRotTime:LREAL:=5;
	
	//RoughTuning
	RotCenter1:vec3;
	BodyPosStart:vec3;
	BodyAngStart:vec3;
	BodyPoseEnd:vec3;
	BodyAngEnd:vec3;
	RoughTuningTime:LREAL:=3;
	RoughTuningExtractTime:LREAL:=2;
	RoughTuningExtendTime:LREAL:=2;
	RoughTuning_FJntRef:ARRAY[0..1] OF vec3;
	RoughTuning_FPosWrtHip:ARRAY[0..1] OF vec3;
	RoughTuning_MJntStart:ARRAY[0..1] OF vec3;
	RoughTuning_MJntRef:ARRAY[0..1] OF vec3;
	RoughTuning_MPosWrtHip:ARRAY[0..1] OF vec3;
	RoughTuning_legPosEnterExtract:ARRAY[0..5] OF vec3;
	
	//FineTuning
	RotCenter2:vec3;
	FineTuning_FJntRef:ARRAY[0..1] OF vec3;
	FineTuning_FPosWrtHip:ARRAY[0..1] OF vec3;
	FineTuningBodyPos:vec3;
	FineTuningBodyAng:vec3;
	realTimeBodyYaw:LREAL;
	realTimeBodyYawLast:lreal;
	
	//LiftMleg
	LiftMleg_MJntStart:ARRAY[0..1] OF vec3;
	LiftMleg_MJntRef:ARRAY[0..1] OF vec3;
	LiftMleg_MPosWrtHip:ARRAY[0..1] OF vec3;
	LiftMlegTime:LREAL:=2;
	
	//SpeedUp
	SpeedUpSubState:UINT:=0;
	SpeedUpAS:UINT:=1;//acceleration
	SpeedUpCS:UINT:=2;//constant velocity
	SpeedUpDS:UINT:=3;//deceleration velocity
	SpeedUpSS:UINT:=4;//stop
	 
	Distance_x_AS:LREAL:=0.3;// acceleration distance in x direction
	Distance_x_DS:LREAL:=0.15;// deceleration distance in x direction
	Distance_y_DS:LREAL:=0.1;// deceleration distance in y direction
	Time_AS:LREAL:=0.3;//acceleration time
	Time_CS:LREAL:=0.05;//constant time
	Time_DS:LREAL:=0.2;//deceleration time
	 
	EnterSpeedUpASCount:UDINT;
	EnterSpeedUpCSCount:UDINT;
	EnterSpeedUpDSCount:UDINT;
	EnterSpeedUpSPCount:UDINT;
	
	SpeedUp_MJntRef:ARRAY[0..1] OF vec3;
	SpeedUp_MPosWrtHip:ARRAY[0..1] OF vec3;
	SpeedUp_FJntRef:ARRAY[0..1] OF vec3;
	SpeedUp_FPosWrtHip:ARRAY[0..1] OF vec3;
	
	body_ref_pos_wrt_body:vec3;
	
	//Slide
	
	//PushReleaseBall
	PushReleaseBall_FJntStart:ARRAY[0..1] OF vec3;
	PushReleaseBall_FPosStartWrtHip:ARRAY[0..1] OF vec3;
	PushReleaseBall_FJntRef:ARRAY[0..1] OF vec3;
	PushReleaseBall_FPosWrtHip:ARRAY[0..1] OF vec3;
	PushTime:LREAL:=0.2;
	PushDistance:LREAL:=0.2;
	DecVelTime:LREAL:=0.1;
	DecVelDistance:LREAL:=0.1;
	PushVelocity:LREAL:=0.5;
	ReleaseTime:LREAL:=0.25;
	
	//SpeedDown
	SpeedDownTime:LREAL:=2;
	SpeedDown_MJntStart:ARRAY[0..1] OF vec3;
	SpeedDown_MJntRef:ARRAY[0..1] OF vec3;
	SpeedDown_MPosWrtHip:ARRAY[0..1] OF vec3;	
	
	//MlegRollC
	MlegRollC_MJntStart:ARRAY[0..1] OF vec3;
	MlegRollC_MPosWrtHip:ARRAY[0..1] OF vec3;
	MlegRollC_MJntRef:ARRAY[0..1] OF vec3;
	MlegRollCTime:LREAL:=3;
	MlegRollC_MJntTarget:ARRAY[0..1,0..2] OF LREAL;
	
	//AddHeight
	AddHeightTime:LREAL:=5;
	AddHeight_FJntStart:ARRAY[0..1] OF vec3;
	AddHeight_FPosWrtHip:ARRAY[0..1] OF vec3;
	
	//FlegRotB
	FlegRotBTime:LREAL:=2;
	FlegRotB_FJntStart:ARRAY[0..1] OF vec3;
	FlegRotB_FJntRef:ARRAY[0..1] OF vec3;
	FlegRotB_FPosWrtHip:ARRAY[0..1] OF vec3;	

END_VAR

METHOD PUBLIC DoPlanning : BOOL
VAR_INPUT
	count : UDINT;
END_VAR
VAR
	i, j  : INT;
END_VAR
IF count = 0 THEN
	isFinished := FALSE;
	Initialize();
END_IF
StateMachine();

TrjPlanning();

IF quit_flag THEN
	isFinished := TRUE;
	quit_flag := FALSE;
END_IF
END_METHOD

METHOD PUBLIC Initialize : BOOL
VAR_INPUT
END_VAR
VAR
	i, j : INT;
	
	leg_pos    : ARRAY[0..2] OF LREAL;
	
	Rb : Mat3;
	hip_pos_j  : Vec3;
	leg_pos_wrt_com : Vec3;
	
END_VAR
Rleg[0]:=SetMat3(1,0,0,0,0,-1,0,1,0);
Rleg[1]:=SetMat3(-1,0,0,0,0,1,0,1,0,);
Rleg[2]:=SetMat3(-1,0,0,0,0,1,0,1,0);
Rleg[3]:=SetMat3(-1,0,0,0,0,1,0,1,0);
Rleg[4]:=SetMat3( -1,0,0,0,0,1,0,1,0);
Rleg[5]:=SetMat3(1,0,0,0,0,-1,0,1,0);

state:=Ready;
RequireMlegRollC:=TRUE;
ReadyFinished:=TRUE;
RequireAddHeight:=FALSE;
RequireFlegRotB:=FALSE;

quit_flag  := FALSE;
gait_cycle := 0;

// control button for each state, need be commented out at actual environment
RequireMlegRollA:=FALSE;
RequireBlegCenter:=FALSE;
RequireFlegRotA:=FALSE;
RequireReduceHeight:=FALSE;	
RequireMlegRollB:=FALSE;	
RequireStoneRot:=FALSE;		
RequireRoughTuning:=FALSE;
RequireFineTuning:=FALSE;
RequireLiftMleg:=FALSE;
RequireSpeedUp:=FALSE;
RequireSlide:=FALSE;
RequirePushReleaseBall:=FALSE;
RequireSpeedDown:=FALSE;
RequireAddHeight:=FALSE;
RequireFlegRotB:=FALSE;
RequireRecoveryReady:=FALSE;

MlegRollAFinished:=FALSE;
BlegCenterFinished:=FALSE;
FlegRotAFinished:=FALSE;
ReduceHeightFinished:=FALSE;
MlegRollBFinished:=FALSE;
StoneRotFinished:=FALSE;
RoughTuningFinished:=FALSE;
FineTuningFinished:=FALSE;
LiftMlegFinished:=FALSE;
SpeedUpFinished:=FALSE;
SlideFinished:=FALSE;
PushReleaseBallFinished:=FALSE;
SpeedDownFinished:=FALSE;
MlegRollCFinished:=FALSE;
AddHeightFinished:=FALSE;
FlegRotBFinished:=FALSE;
RecoveryReadyFinished:=FALSE;
CurlingGaitFinished:=FALSE;

// bodyRot
delta_t:=1.0/gvl.SampleRate;//sample time

//SetTargetValue(GVL.adjust_angle_degree,GVL.target_vel,GVL.stone_rot_vel);
IsReady:=true;

FOR i := 0 TO 5 DO
	FOR j := 0 TO 2 DO
		joint_ref_pos_init[i].data[j] := gvl.jntActualPos[i, j];
		jointPosLast[i,j]:=joint_ref_pos_init[i].data[j];
	END_FOR
END_FOR

sum_height := 0;
FOR j := 0 TO 5 DO
	// FK
	gvl.legCtrl[j].ForwardKinetics(motorAngles := joint_ref_pos_init[j].data, legIndex:=j, tipPosition => leg_pos);
	leg_ref_pos_init_wrt_hip[j] := SetVec3(leg_pos[0], leg_pos[1], leg_pos[2]);
	sum_height := sum_height - leg_ref_pos_init_wrt_hip[j].data[1];
END_FOR
body_ref_pos_init := SetVec3(0, 0, sum_height/6.0);
body_ref_ang_init := SetVec3(0, 0, 0);                            

FOR j := 0 TO 5 DO
	fbRotMat(yaw := body_ref_ang_init.data[2],
             pitch := body_ref_ang_init.data[1],
             roll := body_ref_ang_init.data[0],
             rm => Rb );
	hip_pos_j := SetVec3(hip_pos[j, 0], hip_pos[j, 1], hip_pos[j, 2]);
	leg_pos_wrt_com := VecAdd(MatMulVec(Rleg[j], leg_ref_pos_init_wrt_hip[j]), hip_pos_j);
    leg_ref_pos_init[j] := VecAdd(body_ref_pos_init, MatMulVec(Rb, leg_pos_wrt_com));
END_FOR

body_ref_pos := body_ref_pos_init;
body_ref_ang := body_ref_ang_init;
leg_ref_pos := leg_ref_pos_init;
leg_ref_pos_wrt_hip := leg_ref_pos_init_wrt_hip;

FOR i := 0 TO 5 DO
	FOR j := 0 TO 2 DO
		jointPosTarget[i, j] := joint_ref_pos_init[i].data[j];
		jointVelTarget[i, j] := 0;
		jointFceTarget[i, j] := 0;
	END_FOR
END_FOR
END_METHOD

METHOD PUBLIC StateMachine : BOOL
VAR_INPUT
END_VAR

VAR
	i: INT;
	j: INT;
	RotRadius: LREAL;
END_VAR
IF state=ready  AND RequireMlegRollC=TRUE THEN
	state:=MlegRollC;
	IsReady:=FALSE;
	IsMlegRollC:=TRUE;
	RequireMlegRollC:=FALSE;
	body_ref_pos_enter := body_ref_pos;
	body_ref_ang_enter := body_ref_ang;
	leg_ref_pos_enter := leg_ref_pos;
	EnterMlegRollCCount:=gait_cycle;	
	FOR i:=0 TO 1 DO
		FOR j:=0 TO 2 DO
			MlegRollC_MJntStart[i].data[j]:=jointPosLast[Mapping14[i],j];
		END_FOR
	END_FOR
ELSIF state=MlegRollC AND MlegRollCFinished=TRUE AND RequireAddHeight=TRUE THEN	
	state:=AddHeight;
	RequireAddHeight:=FALSE;
	IsMlegRollC:=FALSE;
	IsAddHeight:=TRUE;
	body_ref_pos_enter := body_ref_pos;
	body_ref_ang_enter := body_ref_ang;
	leg_ref_pos_enter := leg_ref_pos;
	EnterAddHeightCount:=gait_cycle;
	FOR i:=0 TO 1 DO
		FOR j:=0 TO 2 DO
			AddHeight_FJntStart[i].data[j]:=jointPosLast[Mapping23[i],j];
		END_FOR
	END_FOR
	body_target_pos:=body_ref_pos_enter;
	body_target_pos.data[2]:=sum_height/6.0+0.2903;
ELSIF state=AddHeight AND AddHeightFinished=TRUE AND RequireFlegRotB=TRUE THEN	
	state:=FlegRotB;
	IsAddHeight:=FALSE;
	IsFlegRotB:=TRUE;
	RequireFlegRotB:=FALSE;
	body_ref_pos_enter := body_ref_pos;
	body_ref_ang_enter := body_ref_ang;
	leg_ref_pos_enter := leg_ref_pos;
	EnterFlegRotBCount:=gait_cycle;
	FOR i:=0 TO 1 DO
		FOR j:=0 TO 2 DO
			FlegRotB_FJntStart[i].data[j]:=jointPosLast[Mapping23[i],j];
		END_FOR
	END_FOR
ELSIF state=FlegRotB AND FlegRotBFinished=TRUE THEN	
	IsFlegRotB:=FALSE;
	IsCurlingFinished:=TRUE;
	state:=CurlingFinished;
	CurlingGaitFinished:=TRUE;
	quit_flag:=TRUE;
END_IF
END_METHOD

METHOD PUBLIC TrjPlanning : BOOL
VAR_INPUT
END_VAR
VAR
	tr : LREAL;
	i, j : INT;
	Rb : Mat3;
	hip_pos_j : Vec3;
	leg_ref_pos_wrt_com_j : Vec3;
	tmp : Vec3;
	tip_pos, tip_vel : Vec3;
	
	body_ref_pos_start : Vec3;
	body_ref_pos_end : Vec3;
	jointTmpPosLast: ARRAY[0..2] OF LREAL;
	body_ref_ang_start: Vec3;
	leg_ref_pos_start: ARRAY [0..5] OF Vec3;
	leg_ref_pos_target: ARRAY [0..5] OF Vec3;
	body_ref_ang_end: Vec3;
	Rb_target2: Mat3;
	Rb_target1: Mat3;
	leg_ref_pos_end: ARRAY [0..5] OF Vec3;
	fbElipseInterpolation:ElipseInterpolation;
	fbHermitInterpolation:HermitInterpolation;
	holdPos: INT;
END_VAR
gait_cycle := gait_cycle + 1;

IF state=Ready THEN
	body_ref_pos := body_ref_pos_init;
	body_ref_ang := body_ref_ang_init;
	leg_ref_pos := leg_ref_pos_init;
	leg_ref_pos_wrt_hip := leg_ref_pos_init_wrt_hip;
ELSIF state=MlegRollC THEN	
	TrjPlanning_MlegRollC();
ELSIF state=AddHeight THEN	
	TrjPlanning_AddHeight();
ELSIF state=FlegRotB THEN	
	TrjPlanning_FlegRotB();
END_IF

// transform TO leg local frame AND DO inverse kinematics

FOR j := 0 TO 5 DO
	fbRotMat(
    	yaw := body_ref_ang.data[2], 
		pitch := body_ref_ang.data[1], 
		roll := body_ref_ang.data[0], 
		rm => Rb);
	hip_pos_j := SetVec3(hip_pos[j, 0], hip_pos[j, 1], hip_pos[j, 2]);

	//leg_ref_pos_wrt_com = Rb' * (leg_ref_pos - body_ref_pos)
	leg_ref_pos_wrt_com_j := MatMulVec(
		                         MatTranspose(Rb),
								 VecAdd(
									 leg_ref_pos[j],
									 VecNeg(body_ref_pos)
                                 )
                             );
	// leg_ref_pos_wrt_hip = Rleg' * (leg_ref_pos_wrt_com_j - hip_pos)
	leg_ref_pos_next_wrt_hip[j] := MatMulVec(
		                               MatTranspose(Rleg[j]),
									   VecAdd(
										   leg_ref_pos_wrt_com_j,
										   VecNeg(hip_pos_j)
									   )
								   );
								   
	leg_ref_vel_next_wrt_hip[j] := VecMulNum(VecAdd(leg_ref_pos_next_wrt_hip[j], VecNeg(leg_ref_pos_wrt_hip[j])), DINT_TO_LREAL(gvl.sampleRate));
END_FOR


// mapping to actual joints
FOR j := 0 TO 5 DO
	tmp := leg_ref_pos_next_wrt_hip[leg_index_mapping[j]-1];
	tip_pos := SetVec3(tmp.data[0], tmp.data[1], tmp.data[2]);
	tmp := leg_ref_vel_next_wrt_hip[leg_index_mapping[j]-1];
	tip_vel := SetVec3(tmp.data[0], tmp.data[1], tmp.data[2]);
	FOR i:= 0 TO 2 DO
		jointTmpPosLast[i]:=jointPosLast[j,i];
	END_FOR		
	gvl.legCtrl[j].InversePosAndVel(
		tipPos := tip_pos.data, 
		tipVel := tip_vel.data, 
		refPosLast:=jointTmpPosLast,
		legIndex:=j,
		jntPos => joint_ref_pos[j].data, 
		jntVel => joint_ref_vel[j].data);
	
END_FOR

// link to physical outputs
FOR i := 0 TO 5 DO
	FOR j := 0 TO 2 DO
		jointPosTarget[i, j] := joint_ref_pos[i].data[j];
		jointPosLast[i,j]:=jointPosTarget[i, j] ;
		jointVelTarget[i, j] := joint_ref_vel[i].data[j];
		jointFceTarget[i, j] := 0;
	END_FOR
END_FOR

// store refs for next loop
leg_ref_pos_wrt_hip := leg_ref_pos_next_wrt_hip;

IF gait_cycle > tTotalAll * gvl.sampleRate THEN
	quit_flag := TRUE;
END_IF
END_METHOD

METHOD PUBLIC TrjPlanning_AddHeight : BOOL
VAR_INPUT
END_VAR
VAR
	tr: LREAL;
	i: INT;
	Rb_target1: Mat3;
	temp:vec3;
END_VAR
IF  AddHeightFinished=FALSE AND (gait_cycle-EnterAddHeightCount)<=AddHeightTime*gvl.sampleRate THEN
	body_ref_ang:=body_ref_ang_enter;
	leg_ref_pos:=leg_ref_pos_enter;
	tr  := UDINT_TO_LREAL(gait_cycle - EnterAddHeightCount) / gvl.sampleRate / AddHeightTime;
	fbGetPivot(tNow := tr, tTotal := 1.0, pivot => pvt);
	FOR i:=0 TO 2 DO
		body_ref_pos.data[i]:=(1-pvt)*body_ref_pos_enter.data[i]+pvt*body_target_pos.data[i];
	END_FOR
	
	FOR i:=0 TO 1 DO
		gvl.legCtrl[Mapping23[i]].ForwardKinetics(motorAngles:=AddHeight_FJntStart[i].data , legIndex:=Mapping23[i] , tipPosition=>AddHeight_FPosWrtHip[i].data );
		fbRotMat(yaw := body_ref_ang_enter.data[2], pitch := body_ref_ang_enter.data[1],roll := body_ref_ang_enter.data[0], rm => Rb_target1 );
		temp.data[0]:=hip_pos[Mapping23[i],0];temp.data[1]:=hip_pos[Mapping23[i],1];temp.data[2]:=hip_pos[Mapping23[i],2];
		leg_ref_pos[Mapping23[i]]:= VecAdd( MatMulVec(Rb_target1, VecAdd(temp,MatMulVec(Rleg[Mapping23[i]],AddHeight_FPosWrtHip[i]))),body_ref_pos);
	END_FOR
ELSE
	AddHeightFinished:=TRUE;	
	RequireFlegRotB:=TRUE;
END_IF
END_METHOD

METHOD PUBLIC TrjPlanning_FlegRotB : BOOL
VAR_INPUT
END_VAR
VAR
	FlegRotB_FJntState1:ARRAY[0..1,0..2] OF LREAL:=[0*pi/180,162*pi/180,172*pi/180,
                                                    0*pi/180,162*pi/180,172*pi/180];	//side rotates to horizon	
	FlegRotB_FJntState2:ARRAY[0..1,0..2] OF LREAL:=[0*pi/180,162*pi/180,81.588*pi/180,
                                                    0*pi/180,162*pi/180,81.588*pi/180];	;	//shank rotates to rc position
	(*FlegRotB_FJntState3:ARRAY[0..1,0..2] OF LREAL:=[0*pi/180,187.8384*pi/180,81.588*pi/180,
                                                    0*pi/180,187.8384*pi/180,81.588*pi/180];	//thigh rotates to RC position	[-0.3,-0.3209,-0.1246]*)
	FlegRotB_FJntState3:ARRAY[0..1,0..2] OF LREAL:=[0*pi/180,222.0252*pi/180,(254.0072-222.0252)*pi/180,
                                                    0*pi/180,222.0252*pi/180,(254.0072-222.0252)*pi/180];	//thigh rotates to RC position	[-0.3,-0.3209,-0.1246]

																								 									 
	State1Time:LREAL:=2;
	State2Time:LREAL:=2;
	State3Time:LREAL:=2;
	State4Time:LREAL:=2;													 
													 
	tr: lreal;
	i: INT;
	j: INT;
	Rb_target1: Mat3;
	temp: vec3;
END_VAR
IF FlegRotBFinished=FALSE THEN
	IF(gait_cycle-EnterFlegRotBCount)<=State1Time*gvl.sampleRate THEN
		body_ref_pos:=body_ref_pos_enter;
		body_ref_ang:=body_ref_ang_enter;
		leg_ref_pos:=leg_ref_pos_enter;	
		
		tr  := UDINT_TO_LREAL(gait_cycle - EnterFlegRotBCount) / gvl.sampleRate / State1Time;
		fbGetPivot(tNow := tr, tTotal := 1.0, pivot => pvt);	
		FOR i:=0 TO 1 DO
			FOR j:=0 TO 2 DO
				FlegRotB_FJntRef[i].data[j]:=(1-pvt)*FlegRotB_FJntStart[i].data[j]+pvt*(FlegRotB_FJntState1[i,j]);
			END_FOR
			gvl.legCtrl[Mapping23[i]].ForwardKinetics(motorAngles:=FlegRotB_FJntRef[i].data , legIndex:=Mapping23[i] , tipPosition=>FlegRotB_FPosWrtHip[i].data );
			fbRotMat(yaw := body_ref_ang_enter.data[2], pitch := body_ref_ang_enter.data[1],roll := body_ref_ang_enter.data[0], rm =>  Rb_target1 );
			temp.data[0]:=hip_pos[Mapping23[i],0];temp.data[1]:=hip_pos[Mapping23[i],1];temp.data[2]:=hip_pos[Mapping23[i],2];
			leg_ref_pos[Mapping23[i]]:= VecAdd( MatMulVec(Rb_target1, VecAdd(temp,MatMulVec(Rleg[Mapping23[i]],FlegRotB_FPosWrtHip[i]))),body_ref_pos);	
		END_FOR
		
	ELSIF (gait_cycle-EnterFlegRotBCount)<=(State1Time+State2Time)*gvl.sampleRate THEN
		body_ref_pos:=body_ref_pos_enter;
		body_ref_ang:=body_ref_ang_enter;
		leg_ref_pos:=leg_ref_pos_enter;	
		
		tr  := (UDINT_TO_LREAL(gait_cycle - EnterFlegRotBCount) / gvl.sampleRate-State1Time) / State2Time;
		fbGetPivot(tNow := tr, tTotal := 1.0, pivot => pvt);	
		FOR i:=0 TO 1 DO
			FOR j:=0 TO 2 DO
				FlegRotB_FJntRef[i].data[j]:=(1-pvt)*FlegRotB_FJntState1[i,j]+pvt*(FlegRotB_FJntState2[i,j]);
			END_FOR
			gvl.legCtrl[Mapping23[i]].ForwardKinetics(motorAngles:=FlegRotB_FJntRef[i].data , legIndex:=Mapping23[i] , tipPosition=>FlegRotB_FPosWrtHip[i].data );
			fbRotMat(yaw := body_ref_ang_enter.data[2], pitch := body_ref_ang_enter.data[1],roll := body_ref_ang_enter.data[0], rm =>  Rb_target1 );
			temp.data[0]:=hip_pos[Mapping23[i],0];temp.data[1]:=hip_pos[Mapping23[i],1];temp.data[2]:=hip_pos[Mapping23[i],2];
			leg_ref_pos[Mapping23[i]]:= VecAdd( MatMulVec(Rb_target1, VecAdd(temp,MatMulVec(Rleg[Mapping23[i]],FlegRotB_FPosWrtHip[i]))),body_ref_pos);	
		END_FOR	
	ELSIF	(gait_cycle-EnterFlegRotBCount)<=(State1Time+State2Time+State3Time)*gvl.sampleRate THEN
		body_ref_pos:=body_ref_pos_enter;
		body_ref_ang:=body_ref_ang_enter;
		leg_ref_pos:=leg_ref_pos_enter;	
		tr  := (UDINT_TO_LREAL(gait_cycle - EnterFlegRotBCount) / gvl.sampleRate-State1Time-State2Time) / State3Time;
		fbGetPivot(tNow := tr, tTotal := 1.0, pivot => pvt);		
		FOR i:=0 TO 1 DO
			FOR j:=0 TO 2 DO
				FlegRotB_FJntRef[i].data[j]:=(1-pvt)*FlegRotB_FJntState2[i,j]+pvt*(FlegRotB_FJntState3[i,j]);
			END_FOR
			gvl.legCtrl[Mapping23[i]].ForwardKinetics(motorAngles:=FlegRotB_FJntRef[i].data , legIndex:=Mapping23[i] , tipPosition=>FlegRotB_FPosWrtHip[i].data );
			fbRotMat(yaw := body_ref_ang_enter.data[2], pitch := body_ref_ang_enter.data[1],roll := body_ref_ang_enter.data[0], rm =>  Rb_target1 );
			temp.data[0]:=hip_pos[Mapping23[i],0];temp.data[1]:=hip_pos[Mapping23[i],1];temp.data[2]:=hip_pos[Mapping23[i],2];
			leg_ref_pos[Mapping23[i]]:= VecAdd( MatMulVec(Rb_target1, VecAdd(temp,MatMulVec(Rleg[Mapping23[i]],FlegRotB_FPosWrtHip[i]))),body_ref_pos);	
		END_FOR			
	ELSE		
		FlegRotBFinished:=TRUE;
		quit_flag:=true;
	END_IF
END_IF


(*IF FlegRotBFinished=FALSE AND (gait_cycle-EnterFlegRotBCount)<=FlegRotBTime*gvl.sampleRate THEN
	body_ref_pos:=body_ref_pos_enter;
	body_ref_ang:=body_ref_ang_enter;
	leg_ref_pos:=leg_ref_pos_enter;
	
	tr  := UDINT_TO_LREAL(gait_cycle - EnterFlegRotBCount) / gvl.sampleRate / FlegRotBTime;
	fbGetPivot(tNow := tr, tTotal := 1.0, pivot => pvt);
	FOR i:=0 TO 1 DO
		FOR j:=0 TO 2 DO
			FlegRotB_FJntRef[i].data[j]:=(1-pvt)*FlegRotB_FJntStart[i].data[j]+pvt*(FlegRotB_FJntTarget[i,j]);
		END_FOR
		gvl.legCtrl[Mapping23[i]].ForwardKinetics(motorAngles:=FlegRotB_FJntRef[i].data , legIndex:=Mapping23[i] , tipPosition=>FlegRotB_FPosWrtHip[i].data );
		fbRotMat(yaw := body_ref_ang_enter.data[2], pitch := body_ref_ang_enter.data[1],roll := body_ref_ang_enter.data[0], rm =>  Rb_target1 );
		temp.data[0]:=hip_pos[Mapping23[i],0];temp.data[1]:=hip_pos[Mapping23[i],1];temp.data[2]:=hip_pos[Mapping23[i],2];
		leg_ref_pos[Mapping23[i]]:= VecAdd( MatMulVec(Rb_target1, VecAdd(temp,MatMulVec(Rleg[Mapping23[i]],FlegRotB_FPosWrtHip[i]))),body_ref_pos);
	END_FOR
ELSE	
	FlegRotBFinished:=TRUE;
END_IF	*)
END_METHOD

METHOD PUBLIC TrjPlanning_MlegRollC : BOOL
VAR_INPUT
END_VAR
VAR
	MlegRollC_MPosTarget:ARRAY[0..1,0..2] OF LREAL:=[-0.2,-0.1797,-0.1246,
                                                     -0.2,-0.1797,0.1246];
	MlegRollC_MJntTargetRef:ARRAY[0..1,0..2] OF LREAL:=[0,523.2736*pi/180,-235.1052*pi/180,
                                                     0,523.2736*pi/180,-235.1052*pi/180];
	tr: lreal;
	i: INT;
	j: INT;
	Rb_target1: Mat3;
	temp: vec3;
	tempLeg:ARRAY [0..2] OF LREAL;
	tempJnt:ARRAY [0..2] OF LREAL;
	tempRef:ARRAY [0..2] OF LREAL;
END_VAR
IF (gait_cycle-EnterMlegRollCCount)=1 THEN
	FOR i:=0 TO 1 DO
		tempLeg[0]:=MlegRollC_MPosTarget[i,0];tempLeg[1]:=MlegRollC_MPosTarget[i,1];tempLeg[2]:=MlegRollC_MPosTarget[i,2];
		tempRef[0]:=MlegRollC_MJntTargetRef[i,0];tempRef[1]:=MlegRollC_MJntTargetRef[i,1];tempRef[2]:=MlegRollC_MJntTargetRef[i,2];
		GVL.legCtrl[Mapping14[i]].InverseKinetics(tipPosition:=tempLeg , refPosLast:=tempRef , legIndex:=Mapping14[i] , motorAngles=>tempJnt , isSingular=> );
		MlegRollC_MJntTarget[i,0]:=tempJnt[0];MlegRollC_MJntTarget[i,1]:=tempJnt[1];MlegRollC_MJntTarget[i,2]:=tempJnt[2];		
	END_FOR
END_IF

IF MlegRollCFinished=FALSE AND (gait_cycle-EnterMlegRollCCount)<=MlegRollCTime*gvl.sampleRate THEN
	body_ref_pos:=body_ref_pos_enter;
	body_ref_ang:=body_ref_ang_enter;
	leg_ref_pos:=leg_ref_pos_enter;
	
	tr  := UDINT_TO_LREAL(gait_cycle - EnterMlegRollCCount) / gvl.sampleRate / MlegRollCTime;
	fbGetPivot(tNow := tr, tTotal := 1.0, pivot => pvt);
	FOR i:=0 TO 1 DO
		FOR j:=0 TO 2 DO
			MlegRollC_MJntRef[i].data[j]:=(1-pvt)*MlegRollC_MJntStart[i].data[j]+pvt*(MlegRollC_MJntTarget[i,j]);
		END_FOR
		gvl.legCtrl[Mapping14[i]].ForwardKinetics(motorAngles:=MlegRollC_MJntRef[i].data , legIndex:=Mapping14[i] , tipPosition=>MlegRollC_MPosWrtHip[i].data );
		fbRotMat(yaw := body_ref_ang_enter.data[2], pitch := body_ref_ang_enter.data[1],roll := body_ref_ang_enter.data[0], rm =>  Rb_target1 );
		temp.data[0]:=hip_pos[Mapping14[i],0];temp.data[1]:=hip_pos[Mapping14[i],1];temp.data[2]:=hip_pos[Mapping14[i],2];
		leg_ref_pos[Mapping14[i]]:= VecAdd( MatMulVec(Rb_target1, VecAdd(temp,MatMulVec(Rleg[Mapping14[i]],MlegRollC_MPosWrtHip[i]))),body_ref_pos);
	END_FOR	
ELSE	
	MlegRollCFinished:=TRUE;
	RequireAddHeight:=true;
END_IF
END_METHOD

END_FUNCTION_BLOCK

// ---- POUs/GaitPlanner/TrotWalk.TcPOU
FUNCTION_BLOCK TrotWalk
VAR_INPUT
END_VAR
VAR_OUTPUT
END_VAR
VAR
	period:ARRAY [0..1] OF LREAL:=[1,1];//total time of swing and stance
	duty:ARRAY [0..1] OF LREAL:=[0.5,0.5];
	step_height:ARRAY [0..1] OF LREAL:=[0.08,0.08];
	step:ARRAY [0..2] OF LREAL:=[0.1,0.1,0.1];//velocity change step
	delta_t:LREAL:=0.001;//sampling period
	
	(*protect*)
	isFeed : BOOL;
	starveCount : DINT;
	
	// robot geometrical parameters
	hip_pos : ARRAY[0..5, 0..2] OF LREAL := [-0.369,  -0.125, 0,
                                             0,  -0.28, 0,
                                             0.36, -0.125, 0,
                                             0.36, 0.125, 0,
											 0,0.28,0,
											 -0.369,0.125,0];

	leg_index_mapping : ARRAY[0..5] OF INT := [1, 2, 3, 4,5,6];
	Rleg : ARRAY[0..5] OF Mat3;
	Rleg_hip_wrt_trj : ARRAY[0..5] OF Mat3;//髋关节坐标系相对TT轨迹生成坐标系的旋转矩阵，注：TT轨迹生成坐标方位和后腿重合，位置和各腿髋关节原点重合
	
	joint_ref_pos_init : ARRAY[0..5] OF Vec3;
	jointPosLast   : ARRAY[0..5, 0..2] OF LREAL; 
	
	body_ref_pos_init : Vec3;
	body_ref_ang_init : Vec3;
    leg_ref_pos_init : ARRAY[0..5] OF Vec3;
	leg_ref_pos_init_wrt_hip : ARRAY[0..5] OF Vec3;
	
	body_ref_pos : Vec3;
	body_ref_ang : Vec3;
    leg_ref_pos : ARRAY[0..5] OF Vec3;
	leg_ref_pos_wrt_hip : ARRAY[0..5] OF Vec3;
	
	body_ref_pos_next : Vec3;
	body_ref_ang_next : Vec3;
    leg_ref_pos_next : ARRAY[0..5] OF Vec3;
	leg_ref_pos_next_wrt_hip : ARRAY[0..5] OF Vec3;
	leg_ref_vel_next_wrt_hip : ARRAY[0..5] OF Vec3;
	
	// output test
	joint_ref_pos   : ARRAY[0..5] OF Vec3;
	joint_ref_vel   : ARRAY[0..5] OF Vec3;
	
	jointPosTarget  : ARRAY[0..5, 0..2] OF LREAL; 
	jointVelTarget  : ARRAY[0..5, 0..2] OF LREAL;  
	jointFceTarget  : ARRAY[0..5, 0..2] OF LREAL;  
	
	pvt, pvtDot : LREAL;
	
	fbRotmat : RotM;
	fbGetPivot  : GetPivot;
	fbCubicSpline:CubicSpline;
	
	//state
	stance:INT:=1;
	swing:INT:=0;
	ready:INT:=-1;
	init:INT:=-2;
	state:ARRAY[0..1] OF INT:=[-2,-2];
	state_last:ARRAY[0..1] OF INT:=[-1,-1];
	
	gait_cycle : UDINT := 0;
	gait_cycle_enter: array[0..1] of UDINT := [0,0];
	quit_flag : BOOL := FALSE;
	require_stop:BOOL:=FALSE;
	require_move_last:BOOL:=FALSE;
	require_move:BOOL:=FALSE;
	isFinished:BOOL:=FALSE;
	isTrotWalk:bool:=false;
	inTrot: ARRAY [0..1] OF BOOL:=[FALSE,FALSE];
	
	count_en_ST:ARRAY [0..1] OF UDINT:=[0,0];
	count_en_SW:ARRAY [0..1] OF UDINT:=[0,0];
	count_en_RD:ARRAY [0..1] OF UDINT:=[0,0];
	tip_pos_en_ST:ARRAY [0..5] OF vec3;
	tip_pos_en_SW:ARRAY [0..5] OF vec3;
	tip_pos_en_RD:ARRAY [0..5] OF vec3;
	tip_vel_en_ST:ARRAY [0..5] OF vec3;
	tip_vel_en_SW:ARRAY [0..5] OF vec3;
	tip_vel_en_RD:ARRAY [0..5] OF vec3;
	tip_pos_ref:ARRAY [0..5] OF vec3;
	tip_vel_ref:ARRAY [0..5] OF vec3;
	tip_pos_ref_last:ARRAY [0..5] OF vec3;
	
	trot_vel_desire:LREAL:=0;
	side_vel_desire:LREAL:=0;
	turn_rate_desire:LREAL:=0;
	
	trot_vel:ARRAY [0..1] OF LREAL:=[0,0];
	side_vel:ARRAY [0..1] OF LREAL:=[0,0];
	turn_rate:ARRAY [0..1] OF LREAL:=[0,0];
	
	trot_vel_now:ARRAY [0..1] OF LREAL:=[0,0];
	side_vel_now:ARRAY [0..1] OF LREAL:=[0,0];
	turn_vel_now:ARRAY [0..1] OF LREAL:=[0,0];
	
	SwingTrj_tn:ARRAY[0..4] OF LREAL:=[0,0.25,0.5,0.75,1];
	StanceTrj_tn:ARRAY[0..4] OF LREAL:=[0,0.25,0.5,0.75,1];
	ReadyTrj_tn:ARRAY[0..4] OF LREAL:=[0,0.25,0.5,0.75,1];
	
	(*normal_tip_pos_cart:ARRAY[0..5, 0..2] OF LREAL:=[-0.35,-0.3,0,
													 -0.1,-0.3209,0.1246,
													 0.3,-0.3209,0.1246,
													 0.3,-0.3209,-0.1246,
													 -0.1,-0.3209,-0.1246,
													-0.35,-0.3,0];//before change tip	*)	
	normal_tip_pos_cart:ARRAY[0..5, 0..2] OF LREAL:=[-0.35,-0.3209,0,
													 -0.1,-0.3209,0.1246,
													 0.3,-0.3209,0.1246,
													 0.3,-0.3209,-0.1246,
													 -0.1,-0.3209,-0.1246,
													-0.35,-0.3209,0];											
	base_height:LREAL;
	base_x:LREAL;
	base_z:LREAL;
	step_height_now:LREAL;
	step_length_now:LREAL;
	step_side_len_now:LREAL;
	start_height:LREAL;
	Mapping05:ARRAY[0..1] OF INT:=[0,5];
	stopGroup:ARRAY [0..1] OF BOOL:=[FALSE,FALSE];
	flag: INT;
	
	tipForceDesire:ARRAY[0..5,0..2] OF LREAL;
	jntTrqDesire:ARRAY[0..5,0..2] OF LREAL;
	fceLoadTime:LREAL:=0.2;
	tipForceDesireZeros:ARRAY[0..5,0..2] OF LREAL:=[0,0,0,
													 0,0,0,
													 0,0,0,
													 0,0,0,
													 0,0,0,
													 0,0,0];
	tipForceTarget:		 ARRAY[0..5,0..2] OF LREAL:=[0,0,0,
													 0,0,0,
													 0,0,0,
													 0,0,0,
													 0,0,0,
													 0,0,0];
													 
	//posture stabilizer
	bodyRPY : Vec3;		
	lstRollErr: LREAL:=0;
	lstPitchErr: LREAL:=0;
	sumRollErr: LREAL:=0;
	sumPitchErr: LREAL:=0;
	kp:LREAL:=1000;
	ki:LREAL:=3000;//对效果影响较大，kp的1-4倍效果差不多
	kd:LREAL:=100;//和0差别不明显
	kRatio:LREAL:=2;//pitch方向增益要给大点，通过该参数控制
	wrench: Vec3;
	fceStance: Vec3;
	readyToRelease: BOOL;
	enterReadyToReleaseCount:UDINT:=0;
	swingID : ARRAY[0..2] OF DINT;
	stanceID : ARRAY[0..2] OF DINT;
	jntFce : ARRAY[0..5] OF Vec3;
	tipFce : ARRAY[0..5] OF Vec3;//2G
	tipFce2B : ARRAY[0..5] OF Vec3;
	tipFce2H : ARRAY[0..5] OF Vec3;		
	jointFceStartRelease  : ARRAY[0..5, 0..2] OF LREAL;							 
	
END_VAR

METHOD CalcAddfce : BOOL
VAR_INPUT
	//count: UDINT;
END_VAR
VAR_OUTPUT
END_VAR
VAR
	maxAddFce:LREAL;
	maxFceStance:LREAL;
	fmatStance: Mat3;
	//fceStance: Vec3;
	maxFceSwing:LREAL;
	fmatSwing: Mat3;
	fceSwing: Vec3;
	
	rollErr: LREAL;
	pitchErr: LREAL;
	difRollErr: LREAL;
	difPitchErr: LREAL;
	//wrench: Vec3;
	
	tipFceTmp: ARRAY[0..5] OF Vec3;
	ratio: ARRAY[0..5] OF LREAL;
	i: INT;
	j: INT;
	step: LREAL;
	t: LREAL;
	bodyPmx: Mat3;
END_VAR
maxAddFce:=800;
step:=4;
//IF isAllContact=TRUE THEN
//	sumRollErr:=0;
//	sumPitchErr:=0;
//END_IF

rollErr:=bodyRPY.data[0]-gvl.rpy_model[0];
pitchErr:=bodyRPY.data[1]-gvl.rpy_model[1];
IF ABS(rollErr) < 0.002 THEN
	rollErr:=0;
END_IF
IF ABS(pitchErr) < 0.002 THEN
	pitchERr:=0;
END_IF
sumRollErr:=sumRollErr+rollErr*delta_t;
difRollErr:=(rollErr-lstRollErr)/delta_t;
sumPitchErr:=sumPitchErr+pitchErr*delta_t;
difPitchErr:=(pitchErr-lstPitchErr)/delta_t;
lstRollErr:=rollErr;
lstPitchErr:=pitchErr;

wrench.data[0]:=kp*rollErr+ki*sumRollErr+kd*difRollErr;
wrench.data[1]:=kRatio*(kp*pitchErr+ki*sumPitchErr+kd*difPitchErr);
wrench.data[2]:=600;//gravity

//stance leg
fmatStance:=setMat3(leg_ref_pos[stanceID[0]].data[1]-body_ref_pos.data[1],leg_ref_pos[stanceID[1]].data[1]-body_ref_pos.data[1],leg_ref_pos[stanceID[2]].data[1]-body_ref_pos.data[1],
              -leg_ref_pos[stanceID[0]].data[0]+body_ref_pos.data[0],-leg_ref_pos[stanceID[1]].data[0]+body_ref_pos.data[0],-leg_ref_pos[stanceID[2]].data[0]+body_ref_pos.data[0],
              1,1,1);
fceStance:=MatMulVec(inv3(fmatStance),wrench);
maxFceStance:=MAX(ABS(fceStance.data[0]),ABS(fceStance.data[1]),ABS(fceStance.data[2]));
IF maxFceStance>maxAddFce THEN
	FOR i:=0 TO 2 DO
		tipFceTmp[stanceID[i]]:=SetVec3(0,0,-fceStance.data[i]/maxFceStance*maxAddFce);
	END_FOR
ELSE	
	FOR i:=0 TO 2 DO
		tipFceTmp[stanceID[i]]:=SetVec3(0,0,-fceStance.data[i]);
	END_FOR
END_IF
//swing leg
(*fmatSwing:=setMat3(tipPos[swingID[0]].data[1]-bodyPos.data[1],tipPos[swingID[1]].data[1]-bodyPos.data[1],tipPos2B[swingID[2]].data[1]-bodyPos.data[1],
              -tipPos2B[swingID[0]].data[0]+bodyPos.data[0],-tipPos2B[swingID[1]].data[0]+bodyPos.data[0],-tipPos2B[swingID[2]].data[0]+bodyPos.data[0],
              1,1,1);
fceSwing:=MatMulVec(inv3(fmatSwing),wrench);
maxFceSwing:=MAX(ABS(fceSwing.data[0]),ABS(fceSwing.data[1]),ABS(fceSwing.data[2]));
IF maxFceSwing>maxAddFce THEN
	FOR i:=0 TO 2 DO
		tipFceTmp[swingID[i]]:=SetVec3(0,0,-fceSwing.data[i]/maxFceSwing*maxAddFce);
	END_FOR
ELSE	
	FOR i:=0 TO 2 DO
		tipFceTmp[swingID[i]]:=SetVec3(0,0,-fceSwing.data[i]);
	END_FOR
END_IF*)

//方法1,空中给摆动腿加力，感觉只会导致更提前触地，并不能改善倾斜
(*
t := count*deltaT;
IF ABS(t-allContactTime)<deltaT THEN
	FOR i:=0 TO 5 DO
		ratio[i]:=1;
	END_FOR
END_IF
FOR i:=0 TO 2 DO
	IF t-allContactTime<period/2 THEN
		ratio[swingID[i]]:=ratio[swingID[i]]*0.99;//1-0
	ELSE
		ratio[swingID[i]]:=ratio[swingID[i]]/0.99;//0-1
	END_IF
	IF ratio[swingID[i]]>1 THEN//限制在0.01~1
		ratio[swingID[i]]:=1;
	END_IF
	IF ratio[swingID[i]]<0.01 THEN
		ratio[swingID[i]]:=0.01;
	END_IF
	tipFce[stanceID[i]].data[2]:=ratio[stanceID[i]]*tipFceTmp[stanceID[i]].data[2];
	tipFce[swingID[i]].data[2]:=ratio[swingID[i]]*tipFceTmp[swingID[i]].data[2];
END_FOR*)

//方法2
FOR i:=0 TO 2 DO
	IF tipFceTmp[stanceID[i]].data[2]-tipFce[stanceID[i]].data[2]>step THEN
		tipFce[stanceID[i]].data[2]:=tipFce[stanceID[i]].data[2]+step;
	ELSIF tipFceTmp[stanceID[i]].data[2]-tipFce[stanceID[i]].data[2]<-step THEN
		tipFce[stanceID[i]].data[2]:=tipFce[stanceID[i]].data[2]-step;
	ELSE
		tipFce[stanceID[i]].data[2]:=tipFce[stanceID[i]].data[2];
	END_IF
END_FOR

FOR i:=0 TO 2 DO
	tipFce[swingID[i]]:=SetVec3(0,0,tipFce[swingID[i]].data[2]*0.995);
END_FOR


body_ref_ang.data[0]:= gvl.rpy_model[0];
body_ref_ang.data[1]:= gvl.rpy_model[1];                           
body_ref_ang.data[2]:= 0;

leg_ref_pos:=leg_ref_pos_init;
	fbRotMat(yaw := body_ref_ang.data[2], pitch := body_ref_ang.data[1],roll := body_ref_ang.data[0], rm => bodyPmx);
FOR i:=0 TO 5 DO
	tipFce2B[i] := MatMulVec(MatTranspose(bodyPmx),     tipFce[i]);
	tipFce2H[i] := MatMulVec(MatTranspose(Rleg[i]), tipFce2B[i]);
	gvl.legCtrl[i].DesireDriveForce(fTipDes:=tipFce2H[i].data,motorAng:=joint_ref_pos[i].data,
                                    legIndex:=i,fDrvDes=>jntFce[i].data);
END_FOR
END_METHOD

METHOD PUBLIC Cmd2Tgt1Step : lreal
VAR_INPUT
	cmdVel:LREAL;//desired velocity
	curVel:LREAL;//current velocity
	step:LREAL;
END_VAR
VAR_OUTPUT
	trgVel:lreal;
END_VAR
IF step<0 THEN
	step:=-step;
END_IF
IF (curVel-cmdVel)<=-step THEN
    trgVel:=curVel+step;
ELSIF (curVel-cmdVel)>step THEN
    trgVel:=curVel-step;
else
    trgVel:=cmdVel;
END_IF
END_METHOD

METHOD PUBLIC DoPlanning : BOOL
VAR_INPUT
	count : UDINT;
END_VAR
VAR
	i, j  : INT;
END_VAR
IF count = 0 THEN
	isFinished := FALSE;
	Initialize();
END_IF

IF count=10 THEN
	require_move:=TRUE;
END_IF

StateMachine();
TrjPlanning();
//WatchDog(count);//手柄连上再使能

IF quit_flag THEN
	isFinished := TRUE;
	quit_flag := FALSE;
	inTrot[0]:=FALSE;
	inTrot[1]:=FALSE;
	isTrotWalk:=FALSE;
	trot_vel_desire:=0;
	side_vel_desire:=0;
	turn_rate_desire:=0;
	gvl.TrotWalk_trot_vel_desire:=0;
    gvl.TrotWalk_side_vel_desire:=0;
    gvl.TrotWalk_turn_rate_desire:=0;
	FOR i:=0 TO 1 DO
		trot_vel[i]:=0;
		side_vel[i]:=0;
		turn_rate[i]:=0;
	END_FOR
END_IF
END_METHOD

METHOD PUBLIC Initialize : BOOL
VAR_INPUT
END_VAR
VAR
	i, j : INT;
	sum_height : LREAL := 0;
	leg_pos    : ARRAY[0..2] OF LREAL;
	
	Rb : Mat3;
	hip_pos_j  : Vec3;
	leg_pos_wrt_com : Vec3;
	
END_VAR
Rleg[0]:=SetMat3(1,0,0,0,0,-1,0,1,0);
Rleg[1]:=SetMat3(-1,0,0,0,0,1,0,1,0,);
Rleg[2]:=SetMat3(-1,0,0,0,0,1,0,1,0);
Rleg[3]:=SetMat3(-1,0,0,0,0,1,0,1,0);
Rleg[4]:=SetMat3( -1,0,0,0,0,1,0,1,0);
Rleg[5]:=SetMat3(1,0,0,0,0,-1,0,1,0);

Rleg_hip_wrt_trj[0]:=SetMat3(1,0,0,0,1,0,0,0,1);
Rleg_hip_wrt_trj[1]:=SetMat3(-1,0,0,0,1,0,0,0,-1);
Rleg_hip_wrt_trj[2]:=SetMat3(-1,0,0,0,1,0,0,0,-1);
Rleg_hip_wrt_trj[3]:=SetMat3(-1,0,0,0,1,0,0,0,-1);
Rleg_hip_wrt_trj[4]:=SetMat3(-1,0,0,0,1,0,0,0,-1);
Rleg_hip_wrt_trj[5]:=SetMat3(1,0,0,0,1,0,0,0,1);

quit_flag  := FALSE;
gait_cycle := 0;
state[0]:=ready;
state[1]:=ready;
state_last[0]:=init;
state_last[1]:=init;
stopGroup[0]:=FALSE;
stopGroup[1]:=FALSE;
require_move:=FALSE;
require_move_last:=FALSE;
require_stop:=FALSE;
isTrotWalk:=TRUE;

delta_t:=1.0/gvl.sampleRate;

FOR i := 0 TO 5 DO
	FOR j := 0 TO 2 DO
		IF ABS(gvl.jntLastRefPos[i, j] - gvl.jntActualPos[i, j]) < 0.3 THEN
			joint_ref_pos_init[i].data[j] := gvl.jntLastRefPos[i, j];
		ELSE
			joint_ref_pos_init[i].data[j] := gvl.jntActualPos[i, j];
		END_IF
		jointPosLast[i,j]:=joint_ref_pos_init[i].data[j];
	END_FOR
END_FOR

sum_height := 0;
FOR j := 0 TO 5 DO
	// FK
	gvl.legCtrl[j].ForwardKinetics(motorAngles := joint_ref_pos_init[j].data, legIndex:=j, tipPosition => leg_pos);
	leg_ref_pos_init_wrt_hip[j] := SetVec3(leg_pos[0], leg_pos[1], leg_pos[2]);
	sum_height := sum_height - leg_ref_pos_init_wrt_hip[j].data[1];
END_FOR
body_ref_pos_init := SetVec3(0, 0, sum_height/6.0);
body_ref_ang_init := SetVec3(0, 0, 0);

bodyRPY.data[0]:= gvl.rpy_model[0];
bodyRPY.data[1]:= gvl.rpy_model[1];                           
bodyRPY.data[2]:= 0;

FOR j := 0 TO 5 DO
	fbRotMat(yaw := body_ref_ang_init.data[2],
             pitch := body_ref_ang_init.data[1],
             roll := body_ref_ang_init.data[0],
             rm => Rb );
	hip_pos_j := SetVec3(hip_pos[j, 0], hip_pos[j, 1], hip_pos[j, 2]);
	leg_pos_wrt_com := VecAdd(MatMulVec(Rleg[j], leg_ref_pos_init_wrt_hip[j]), hip_pos_j);
    leg_ref_pos_init[j] := VecAdd(body_ref_pos_init, MatMulVec(Rb, leg_pos_wrt_com));
END_FOR

FOR i:=0 TO 5 DO
	tip_vel_ref[i]:=setVec3(0,0,0);
	tip_pos_ref[i]:= MatMulVec( Rleg_hip_wrt_trj[i], leg_ref_pos_init_wrt_hip[i]);
	FOR j:=0 TO 2 DO
		normal_tip_pos_cart[i,j]:=tip_pos_ref[i].data[j];
	END_FOR
END_FOR
tip_pos_ref_last:=tip_pos_ref;

body_ref_pos := body_ref_pos_init;
body_ref_ang := body_ref_ang_init;
leg_ref_pos := leg_ref_pos_init;
leg_ref_pos_wrt_hip := leg_ref_pos_init_wrt_hip;

FOR i := 0 TO 5 DO
	FOR j := 0 TO 2 DO
		jointPosTarget[i, j] := joint_ref_pos_init[i].data[j];
		jointVelTarget[i, j] := 0;
		jointFceTarget[i, j] := 0;
	END_FOR
	tipFce[i]:=SetVec3(0,0,0);
END_FOR

stanceID[0]:=1;stanceID[1]:=3;stanceID[2]:=5;
swingID[0]:=0;swingID[1]:=2;swingID[2]:=4;

enterReadyToReleaseCount:=0;
lstRollErr:=0;
lstPitchErr:=0;
sumRollErr:=0;
sumPitchErr:=0;
readyToRelease:=FALSE;
END_METHOD

METHOD PUBLIC StateMachine : BOOL
VAR_INPUT
END_VAR
VAR
	temp:LREAL;
	i: INT;
	j: INT;
	k: INT;
END_VAR
//set target value
trot_vel_desire:=gvl.TrotWalk_trot_vel_desire;
side_vel_desire:=gvl.TrotWalk_side_vel_desire;
turn_rate_desire:=gvl.TrotWalk_turn_rate_desire;
step[0]:=gvl.TrotWalk_step[0];
step[1]:=gvl.TrotWalk_step[1];
step[2]:=gvl.TrotWalk_step[2];

//state switch
IF require_move_last=FALSE AND require_move=TRUE THEN
	gait_cycle_enter[0]:=gait_cycle;
	gait_cycle_enter[1]:=gait_cycle;
	require_move:=FALSE;
	flag:=1;
	FOR i:=0 TO 1 DO
		inTrot[i]:=TRUE;
		stopGroup[i]:=FALSE;
		duty[i]:=gvl.duty_desire;
		period[i]:=gvl.period_desire;
		step_height[i]:=gvl.step_height_desire;
	END_FOR
END_IF
IF inTrot[0]=TRUE THEN
	temp:=(gait_cycle-gait_cycle_enter[0]) MOD TRUNC(period[0]*gvl.sampleRate);
	IF temp>=(1-duty[0])*gvl.sampleRate*period[0] THEN
		state[0]:=stance;
	ELSE 
		state[0]:=swing;
	END_IF
END_IF
IF inTrot[1]=TRUE THEN	
	IF flag=1 THEN
		temp:=TRUNC((gait_cycle-gait_cycle_enter[1]+0.5*period[1]*gvl.sampleRate) )MOD TRUNC(period[1]*gvl.sampleRate);
	ELSE
		temp:=TRUNC((gait_cycle-gait_cycle_enter[1]) )MOD TRUNC(period[1]*gvl.sampleRate);
	END_IF
	
	(*IF temp>=(1-duty[1])*gvl.sampleRate*period[1] THEN
		state[1]:=stance;
	ELSE 
		state[1]:=swing;			
	END_IF*)
	
	IF state[1]=ready AND (gait_cycle-gait_cycle_enter[0])<LREAL_TO_UDINT(0.5*period[0]*gvl.sampleRate) AND flag=1 THEN
		state[1]:=ready;
	ELSE
		flag:=0;
		IF temp>=(1-duty[1])*gvl.sampleRate*period[1] THEN
			state[1]:=stance;
		ELSE 
			state[1]:=swing;			
		END_IF
	END_IF
END_IF

FOR i:=0 TO 1 DO
	IF state[i]<> state_last[i] THEN
		IF state[i]=stance THEN
			count_en_ST[i]:=gait_cycle;
			IF i=0 THEN
				stanceID[0]:=0;stanceID[1]:=2;stanceID[2]:=4;
			END_IF
			IF i=1 THEN
				stanceID[0]:=1;stanceID[1]:=3;stanceID[2]:=5;
			END_IF
			
			FOR j:=0 TO 2 DO
				FOR k:=0 TO 2 DO
					tip_pos_en_ST[2*j+i].data[k]:=tip_pos_ref[2*j+i].data[k];
					tip_vel_en_ST[2*j+i].data[k]:=tip_vel_ref[2*j+i].data[k];
				END_FOR
			END_FOR
		END_IF
		
		IF state[i]=swing THEN
			count_en_SW[i]:=gait_cycle;
			IF i=0 THEN
				swingID[0]:=0;swingID[1]:=2;swingID[2]:=4;
			END_IF
			IF i=1 THEN
				swingID[0]:=1;swingID[1]:=3;swingID[2]:=5;
			END_IF			
			
			gait_cycle_enter[i]:=gait_cycle;
			FOR j:=0 TO 2 DO
				FOR k:=0 TO 2 DO
					tip_pos_en_SW[2*j+i].data[k]:=tip_pos_ref[2*j+i].data[k];
					tip_vel_en_SW[2*j+i].data[k]:=tip_vel_ref[2*j+i].data[k];
				END_FOR
			END_FOR	
			duty[i]:=gvl.duty_desire;
			period[i]:=gvl.period_desire;
			step_height[i]:=gvl.step_height_desire;
			IF 	require_stop=TRUE THEN
				trot_vel_desire:=0;
				side_vel_desire:=0;
				turn_rate_desire:=0;
				gvl.TrotWalk_trot_vel_desire:=0;
                gvl.TrotWalk_side_vel_desire:=0;
                gvl.TrotWalk_turn_rate_desire:=0;
								
				IF trot_vel_desire=trot_vel[i] AND side_vel_desire=side_vel[i] AND turn_rate_desire=turn_rate[i] THEN	
					state[i]:=ready;
					stopGroup[i]:=TRUE;
					inTrot[i]:=FALSE;
				END_IF
			END_IF
			Cmd2Tgt1Step(cmdVel:= trot_vel_desire, curVel:=trot_vel[i] , step:= step[0], trgVel=>trot_vel[i] );
			Cmd2Tgt1Step(cmdVel:= side_vel_desire, curVel:=side_vel[i] , step:= step[1], trgVel=>side_vel[i] );
			Cmd2Tgt1Step(cmdVel:= turn_rate_desire, curVel:=turn_rate[i] , step:= step[2], trgVel=>turn_rate[i] );
		END_IF
		
		IF state[i]=ready THEN
			count_en_RD[i]:=gait_cycle;
			FOR j:=0 TO 2 DO
				FOR k:=0 TO 2 DO
					tip_pos_en_RD[2*j+i].data[k]:=tip_pos_ref[2*j+i].data[k];
					tip_vel_en_RD[2*j+i].data[k]:=tip_vel_ref[2*j+i].data[k];
				END_FOR
			END_FOR			
		END_IF
	END_IF
	IF state[i]=ready AND gait_cycle-count_en_RD[i]=LREAL_TO_UDINT(2*gvl.sampleRate) THEN	
		count_en_RD[i]:=gait_cycle;
		FOR j:=0 TO 2 DO
			FOR k:=0 TO 2 DO
				tip_pos_en_RD[2*j+i].data[k]:=tip_pos_ref[2*j+i].data[k];
				tip_vel_en_RD[2*j+i].data[k]:=tip_vel_ref[2*j+i].data[k];
			END_FOR
		END_FOR			
	END_IF		
END_FOR

IF stopGroup[0]=TRUE AND stopGroup[1]=TRUE AND require_stop=TRUE AND readyToRelease=FALSE  THEN
	require_stop:=FALSE;
	readyToRelease:=TRUE;
	enterReadyToReleaseCount:=gait_cycle;
	isTrotWalk:=FALSE;
	jointFceStartRelease:=jointFceTarget;
END_IF


state_last:=state; 
require_move_last:=require_move;
END_METHOD

METHOD PUBLIC TrjPlanning : BOOL
VAR_INPUT
END_VAR

VAR
	i: INT;
	k:int;
	FixTrj_tn:ARRAY[0..4] OF LREAL:=[0,0.25,0.5,0.75,1];
	InterplateValue:ARRAY[0..4] OF LREAL;
	InterplateTime:ARRAY[0..4] OF LREAL;
	start_vel:LREAL;
	end_vel:LREAL;
	j: INT;
	Rb_target1: Mat3;
	temp: vec3;
	Rb: Mat3;
	
	hip_pos_j : Vec3;
	leg_ref_pos_wrt_com_j : Vec3;
	tmp : Vec3;
	tip_pos, tip_vel : Vec3;
	jointTmpPosLast: ARRAY[0..2] OF LREAL;
	
	tipForceDesireLegA:	 ARRAY[0..5,0..2] OF LREAL:=[0,-125*0,0,
													 0,0,0,
													 0,0,0,
													 0,0,0,
													 0,0,0,
													 0,0,0];
	tipForceDesireLegF:	 ARRAY[0..5,0..2] OF LREAL:=[0,0,0,
													 0,0,0,
													 0,0,0,
													 0,0,0,
													 0,0,0,
													 0,-145*0.3,0];
	tr: LREAL;
	
	tempTipForce:ARRAY [0..2] OF LREAL;
	temJntActPos:ARRAY [0..2] OF LREAL;
	tempDesJntTrq:ARRAY [0..2] OF LREAL;
END_VAR
gait_cycle := gait_cycle + 1;
FOR k:=0 TO 1 DO
	IF state[k]=swing THEN
		FOR i:=0 TO 4 DO
			SwingTrj_tn[i]:=FixTrj_tn[i]*period[k]*(1-duty[k]);
		END_FOR
		step_height_now :=step_height[k];
		FOR i:=0 TO 2 DO
			//trj planning in y direction (up/down)
			base_height:=normal_tip_pos_cart[2*i+k,1];
			start_height:=tip_pos_en_SW[2*i+k].data[1];
			InterplateValue[0]:=start_height;
			InterplateValue[1]:=(base_height * 0.05 + start_height * 0.95) + step_height_now * 0.6;
			InterplateValue[2]:=(base_height * 0.25 + start_height * 0.75) + step_height_now * 1.0;
			InterplateValue[3]:=(base_height * 0.65 + start_height * 0.35) + step_height_now * 0.6;
			InterplateValue[4]:=base_height;	
			end_vel:=-0.01 / (period[k] * duty[k]);		
			start_vel:=tip_vel_en_SW[2*i+k].data[1];
			fbCubicSpline(x:=SwingTrj_tn , y:=InterplateValue , dy0:=start_vel , dy4:=end_vel , 
				xt:=(gait_cycle-count_en_SW[k])*delta_t , yt=> tip_pos_ref[2*i+k].data[1], vt=> );
				
			//trj planning in x direction (forward/backward)
			base_x:=normal_tip_pos_cart[2*i+k,0];
			trot_vel_now[k]:=trot_vel[k]-turn_rate[k]*(hip_pos[2*i+k,1]-normal_tip_pos_cart[2*i+k,2]);
			step_length_now:= period[k] * duty[k] * trot_vel_now[k];
		 	InterplateValue[0]:=tip_pos_en_SW[2*i+k].data[0];	
		 	InterplateValue[1]:=base_x-0.48*step_length_now;;
		 	InterplateValue[2]:=base_x;
		 	InterplateValue[3]:=base_x+0.48*step_length_now;
		 	InterplateValue[4]:=base_x+0.5*step_length_now;
		 	end_vel:=-trot_vel_now[k];
		 	start_vel:=tip_vel_en_SW[2*i+k].data[0];
			fbCubicSpline(x:=SwingTrj_tn , y:=InterplateValue , dy0:=start_vel , dy4:=end_vel , 
				xt:=(gait_cycle-count_en_SW[k])*delta_t , yt=> tip_pos_ref[2*i+k].data[0], vt=> );			
			
			//trj planning in z direction (right/left)
			base_z:=normal_tip_pos_cart[2*i+k,2];
			turn_vel_now[k]:=turn_rate[k]*(hip_pos[2*i+k,0]+normal_tip_pos_cart[2*i+k,0])+side_vel[k];
			step_side_len_now := period[k] * duty[k] * turn_vel_now[k];
			InterplateValue[0]:=tip_pos_en_SW[2*i+k].data[2];
		 	InterplateValue[1]:=base_z+0.48* step_side_len_now;
		 	InterplateValue[2]:=base_z;
		 	InterplateValue[3]:=base_z-0.48* step_side_len_now;
		 	InterplateValue[4]:=base_z-0.50* step_side_len_now;			
			end_vel:=turn_vel_now[k];
		 	start_vel:=tip_vel_en_SW[2*i+k].data[2];			
		 	fbCubicSpline(x:=SwingTrj_tn , y:=InterplateValue , dy0:=start_vel , dy4:=end_vel , 
				xt:=(gait_cycle-count_en_SW[k])*delta_t , yt=> tip_pos_ref[2*i+k].data[2], vt=> );				
		END_FOR
	ELSIF state[k]=stance THEN 
		FOR i:=0 TO 4 DO
			StanceTrj_tn[i]:=FixTrj_tn[i]*period[k]*duty[k];
		END_FOR
		FOR i:=0 TO 2 DO
			//force compensator
			IF k=0 THEN
				tipForceTarget:=tipForceDesireLegA;
			ELSE
				tipForceTarget:=tipForceDesireLegF;
			END_IF
			IF gait_cycle-count_en_ST[k]>=0 AND  (gait_cycle-count_en_ST[k])<=fceLoadTime*gvl.sampleRate THEN
				tr  := UDINT_TO_LREAL(gait_cycle-count_en_ST[k]) / gvl.sampleRate / fceLoadTime;
				fbGetPivot(tNow := tr, tTotal := 1.0, pivot => pvt);
				FOR j:=0 TO 2 DO
					tipForceDesire[2*i+k,j]:=(1-pvt)*tipForceDesireZeros[2*i+k,j]+pvt*tipForceTarget[2*i+k,j];
				END_FOR
			ELSIF gait_cycle-count_en_ST[k]>=LREAL_TO_UDINT((period[k]*duty[k]-fceLoadTime)*gvl.sampleRate) AND gait_cycle-count_en_ST[k]<=LREAL_TO_UDINT(period[k]*duty[k]*gvl.sampleRate) THEN
				FOR j:=0 TO 2 DO
					tipForceDesire[2*i+k,j]:=(1-pvt)*tipForceTarget[2*i+k,j]+pvt*tipForceDesireZeros[2*i+k,j];
				END_FOR
			END_IF 

			//trj planning in y direction (up/down)
			start_height:=tip_pos_en_ST[2*i+k].data[1];
			InterplateValue[0]:=start_height;
			InterplateValue[1]:=start_height-0.0045*0;//*0.1
			InterplateValue[2]:=start_height-0.0085*0;
			InterplateValue[3]:=start_height-0.0125*0;
			InterplateValue[4]:=start_height-0.0160*0;			
			end_vel:=0;
			start_vel:=tip_vel_en_ST[2*i+k].data[1];
			fbCubicSpline(x:=StanceTrj_tn , y:=InterplateValue , dy0:=start_vel , dy4:=end_vel , 
				xt:=(gait_cycle-count_en_ST[k])*delta_t , yt=> tip_pos_ref[2*i+k].data[1], vt=> );	
			
		    //trj planning in X direction (forward/backward)
			trot_vel_now[k]:=trot_vel[k]-turn_rate[k]*(hip_pos[2*i+k,1]-normal_tip_pos_cart[2*i+k,2]);	
			step_length_now := period[k] * duty[k] * trot_vel_now[k];
			InterplateValue[0]:=tip_pos_en_ST[2*i+k].data[0];
			InterplateValue[1]:=tip_pos_en_ST[2*i+k].data[0]-0.28*step_length_now;
			InterplateValue[2]:=tip_pos_en_ST[2*i+k].data[0]-0.50*step_length_now;
			InterplateValue[3]:=tip_pos_en_ST[2*i+k].data[0]-0.72*step_length_now;
			InterplateValue[4]:=tip_pos_en_ST[2*i+k].data[0]-1.00*step_length_now;	
			end_vel:= -trot_vel_now[k];
			start_vel:=tip_vel_en_ST[2*i+k].data[0];		
			fbCubicSpline(x:=StanceTrj_tn , y:=InterplateValue , dy0:=start_vel , dy4:=end_vel , 
				xt:=(gait_cycle-count_en_ST[k])*delta_t , yt=> tip_pos_ref[2*i+k].data[0], vt=> );
			
			// trj planning in z direction (right/left)
			turn_vel_now[k]:=turn_rate[k]*(hip_pos[2*i+k,0]+normal_tip_pos_cart[2*i+k,0])+side_vel[k];
			step_side_len_now := period[k] * duty[k] * turn_vel_now[k];
			InterplateValue[0]:=tip_pos_en_ST[2*i+k].data[2];
			InterplateValue[1]:=tip_pos_en_ST[2*i+k].data[2]+0.28*step_side_len_now;
			InterplateValue[2]:=tip_pos_en_ST[2*i+k].data[2]+0.50*step_side_len_now;
			InterplateValue[3]:=tip_pos_en_ST[2*i+k].data[2]+0.72*step_side_len_now;
			InterplateValue[4]:=tip_pos_en_ST[2*i+k].data[2]+1.00*step_side_len_now;
			end_vel:=turn_vel_now[k];
			start_vel:=tip_vel_en_ST[2*i+k].data[2];
			fbCubicSpline(x:=StanceTrj_tn , y:=InterplateValue , dy0:=start_vel , dy4:=end_vel , 
				xt:=(gait_cycle-count_en_ST[k])*delta_t , yt=> tip_pos_ref[2*i+k].data[2], vt=> );				
		END_FOR
	ELSE	
		FOR i:=0 TO 4 DO
			ReadyTrj_tn[i]:=FixTrj_tn[i]*2;//2s for ready gait
		END_FOR	
		FOR i:=0 TO 2 DO
			//trj planning in x direction (forward/backward)
			InterplateValue[0]:=tip_pos_en_RD[2*i+k].data[0];
			InterplateValue[1]:=tip_pos_en_RD[2*i+k].data[0];
			InterplateValue[2]:=tip_pos_en_RD[2*i+k].data[0];
			InterplateValue[3]:=tip_pos_en_RD[2*i+k].data[0];
			InterplateValue[4]:=tip_pos_en_RD[2*i+k].data[0];
			end_vel:=0;
			start_vel:=tip_vel_en_ST[2*i+k].data[0];
			fbCubicSpline(x:=ReadyTrj_tn , y:=InterplateValue , dy0:=start_vel , dy4:=end_vel , 
				xt:=(gait_cycle-count_en_RD[k])*delta_t , yt=> tip_pos_ref[2*i+k].data[0], vt=> );	
			
			//trj planning in y direction (right/left)
			InterplateValue[0]:=tip_pos_en_RD[2*i+k].data[1];
			InterplateValue[1]:=tip_pos_en_RD[2*i+k].data[1];
			InterplateValue[2]:=tip_pos_en_RD[2*i+k].data[1];
			InterplateValue[3]:=tip_pos_en_RD[2*i+k].data[1];
			InterplateValue[4]:=tip_pos_en_RD[2*i+k].data[1];
			end_vel:=0;
			start_vel:=tip_vel_en_ST[2*i+k].data[1];
			fbCubicSpline(x:=ReadyTrj_tn , y:=InterplateValue , dy0:=start_vel , dy4:=end_vel , 
				xt:=(gait_cycle-count_en_RD[k])*delta_t , yt=> tip_pos_ref[2*i+k].data[1], vt=> );				
		
			//trj planning in z direction (up/down)
			InterplateValue[0]:=tip_pos_en_RD[2*i+k].data[2];
			InterplateValue[1]:=tip_pos_en_RD[2*i+k].data[2];
			InterplateValue[2]:=tip_pos_en_RD[2*i+k].data[2];
			InterplateValue[3]:=tip_pos_en_RD[2*i+k].data[2];
			InterplateValue[4]:=tip_pos_en_RD[2*i+k].data[2];
			end_vel:=0;
			start_vel:=tip_vel_en_ST[2*i+k].data[2];
			fbCubicSpline(x:=ReadyTrj_tn , y:=InterplateValue , dy0:=start_vel , dy4:=end_vel , 
				xt:=(gait_cycle-count_en_RD[k])*delta_t , yt=> tip_pos_ref[2*i+k].data[2], vt=> );				
		END_FOR
	END_IF
END_FOR

FOR i:=0 TO 5 DO
	FOR j:=0 TO 2 DO
		tip_vel_ref[i].data[j]:=(tip_pos_ref[i].data[j]-tip_pos_ref_last[i].data[j])/delta_t;
	END_FOR
END_FOR
tip_pos_ref_last:=tip_pos_ref;

body_ref_pos:=body_ref_pos_init;
//body_ref_ang:=body_ref_ang_init;

body_ref_ang.data[0]:= gvl.rpy_model[0];
body_ref_ang.data[1]:= gvl.rpy_model[1];                           
body_ref_ang.data[2]:= 0;

leg_ref_pos:=leg_ref_pos_init;
FOR i:=0 TO 5 DO
	fbRotMat(yaw := body_ref_ang.data[2], pitch := body_ref_ang.data[1],roll := body_ref_ang.data[0], rm =>  Rb_target1 );
	temp.data[0]:=hip_pos[i,0];temp.data[1]:=hip_pos[i,1];temp.data[2]:=hip_pos[i,2];
	leg_ref_pos[i]:= VecAdd( MatMulVec(Rb_target1, VecAdd(temp,MatMulVec(Rleg[0],tip_pos_ref[i]))),body_ref_pos);
END_FOR

// transform TO leg local frame AND DO inverse kinematics

FOR j := 0 TO 5 DO
	fbRotMat(
    	yaw := body_ref_ang.data[2], 
		pitch := body_ref_ang.data[1], 
		roll := body_ref_ang.data[0], 
		rm => Rb);
	hip_pos_j := SetVec3(hip_pos[j, 0], hip_pos[j, 1], hip_pos[j, 2]);

	//leg_ref_pos_wrt_com = Rb' * (leg_ref_pos - body_ref_pos)
	leg_ref_pos_wrt_com_j := MatMulVec(
		                         MatTranspose(Rb),
								 VecAdd(
									 leg_ref_pos[j],
									 VecNeg(body_ref_pos)
                                 )
                             );
	// leg_ref_pos_wrt_hip = Rleg' * (leg_ref_pos_wrt_com_j - hip_pos)
	leg_ref_pos_next_wrt_hip[j] := MatMulVec(
		                               MatTranspose(Rleg[j]),
									   VecAdd(
										   leg_ref_pos_wrt_com_j,
										   VecNeg(hip_pos_j)
									   )
								   );
								   
	leg_ref_vel_next_wrt_hip[j] := VecMulNum(VecAdd(leg_ref_pos_next_wrt_hip[j], VecNeg(leg_ref_pos_wrt_hip[j])), DINT_TO_LREAL(gvl.sampleRate));
END_FOR


// mapping to actual joints
FOR j := 0 TO 5 DO
	tmp := leg_ref_pos_next_wrt_hip[leg_index_mapping[j]-1];
	tip_pos := SetVec3(tmp.data[0], tmp.data[1], tmp.data[2]);
	tmp := leg_ref_vel_next_wrt_hip[leg_index_mapping[j]-1];
	tip_vel := SetVec3(tmp.data[0], tmp.data[1], tmp.data[2]);
	FOR i:= 0 TO 2 DO
		jointTmpPosLast[i]:=jointPosLast[j,i];
	END_FOR		
	gvl.legCtrl[j].InversePosAndVel(
		tipPos := tip_pos.data, 
		tipVel := tip_vel.data, 
		refPosLast:=jointTmpPosLast,
		legIndex:=j,
		jntPos => joint_ref_pos[j].data, 
		jntVel => joint_ref_vel[j].data);
	
END_FOR

// link to physical outputs
FOR i := 0 TO 5 DO
	FOR j := 0 TO 2 DO
		jointPosTarget[i, j] := joint_ref_pos[i].data[j];
		jointPosLast[i,j]:=jointPosTarget[i, j] ;
		jointVelTarget[i, j] := joint_ref_vel[i].data[j];
		jointFceTarget[i, j] := 0;
	END_FOR
END_FOR



IF isTrotWalk=TRUE THEN
	
	FOR i:=0 TO 5 DO
		tempTipForce[0]:=tipForceDesire[i,0];tempTipForce[1]:=tipForceDesire[i,1];tempTipForce[2]:=tipForceDesire[i,2];
		temJntActPos[0]:=gvl.jntActualPos[i,0];temJntActPos[1]:=gvl.jntActualPos[i,1];temJntActPos[2]:=gvl.jntActualPos[i,2];
		gvl.legCtrl[i].DesireDriveForce(fTipDes:=tempTipForce , motorAng:=temJntActPos , legIndex:=i , fDrvDes=>tempDesJntTrq );
		jntTrqDesire[i,0]:=tempDesJntTrq[0];jntTrqDesire[i,1]:=tempDesJntTrq[1];jntTrqDesire[i,2]:=tempDesJntTrq[2];
	END_FOR

	CalcAddfce();
	FOR i := 0 TO 5 DO
		FOR j := 0 TO 2 DO
			//jointFceTarget[i, j] := jntFce[i].data[j];//姿态稳定器
			jointFceTarget[i, j] := jntFce[i].data[j]+jntTrqDesire[i,j];//姿态稳定器+静态补偿
		END_FOR
	END_FOR	
END_IF
IF readyToRelease=TRUE THEN//use 100 count to release
	FOR i := 0 TO 5 DO
		FOR j := 0 TO 2 DO
			jointFceTarget[i, j] := jointFceStartRelease[i, j]-0.01*(gait_cycle-enterReadyToReleaseCount)*jointFceStartRelease[i,j];
		END_FOR
	END_FOR
	IF gait_cycle*delta_T-enterReadyToReleaseCount*delta_T>=100*delta_T THEN
		quit_flag:=TRUE;
		readyToRelease:=FALSE;
	END_IF
END_IF


// store refs for next loop
leg_ref_pos_wrt_hip := leg_ref_pos_next_wrt_hip;
END_METHOD

METHOD WatchDog : BOOL
VAR_INPUT
	count: UDINT;
END_VAR
IF isFeed=TRUE THEN//可能是通过手柄控制该变量，固定周期发送一次true过来，因该更新周期小于0.5s。假如固定周期内没有发送true过来，计时超过0.5s后程序将改变步长为零
	starveCount := count + TRUNC(gvl.sampleRate*0.5);//0.5 second
	isFeed := FALSE;
END_IF

IF count>=starveCount THEN
	gvl.TrotWalk_trot_vel_desire:=0;
    gvl.TrotWalk_side_vel_desire:=0;
    gvl.TrotWalk_turn_rate_desire:=0;
END_IF
END_METHOD

END_FUNCTION_BLOCK

// ---- POUs/GaitPlanner/WalkSlopeGait.TcPOU
FUNCTION_BLOCK WalkSlopeGait
VAR_INPUT
END_VAR
VAR_OUTPUT
END_VAR
VAR
	(*cmd var*)
	period : LREAL := 1;
	cmdH : LREAL := 0.15;
	cmdL : LREAL := 0;
	cmdLa : LREAL := 0;
	cmdYaw : LREAL := 0;
	isLastStep : BOOL := FALSE;
	swingDir : INT := 0;
	(*protect*)
	isFeed : BOOL;
	starveCount : DINT;
	
	(*general essential var*)
	hipPos2B : ARRAY[0..5] OF Vec3;
	hipPmx2B : ARRAY[0..5] OF Mat3;//wrt body
	objRotMtx : RotM;
	
	jntPosInit : ARRAY[0..5] OF Vec3;
	bodyPosInit : Vec3;
	bodyRPYInit : Vec3;
	bodyPmxInit : Mat3;
	tipPosInit   : ARRAY[0..5] OF Vec3;
	tipPosInit2H : ARRAY[0..5] OF Vec3;
	tipPosInit2B : ARRAY[0..5] OF Vec3;//recover tip pos
	bodyPos : Vec3;
	bodyRPY : Vec3;
	tipPos   : ARRAY[0..5] OF Vec3;
	tipPos2H : ARRAY[0..5] OF Vec3;
	bodyRefH : LREAL;
	
	jointPosTarget  : ARRAY[0..5, 0..2] OF LREAL; 
	jointVelTarget  : ARRAY[0..5, 0..2] OF LREAL;  
	jointFceTarget  : ARRAY[0..5, 0..2] OF LREAL;
	isFinished : BOOL;
	(*end of general essential var*)
	
	(*specific var in this gait*)
	bodyPosInit2T : Vec3;
	bodyPosTrgt : Vec3;
	bodyRPYTrgt : Vec3;
	bodyPmxTrgt : Mat3;
	bodyPmx : Mat3;
	bodyVelInit : Vec3;
	bodyVelInit2T : Vec3;
	bodyVelTrgt2T : Vec3;
	bodyOmgInit : LREAL;
	bodyOmgTrgt : LREAL;
	tipPosTrgt : ARRAY[0..5] OF Vec3;
	tipPosTrgt2T : ARRAY[0..5] OF Vec3;
	tipPos2B : ARRAY[0..5] OF Vec3;
	tipPosTrgtBase : ARRAY[0..5] OF Vec3;
	
	bodyPos2T : Vec3;
	bodyVel : Vec3;
	bodyVel2T : Vec3;
	bodyOmg : LREAL;
	tipVel : ARRAY[0..5] OF Vec3;
	jntPos   : ARRAY[0..5] OF Vec3;
	jntVel   : ARRAY[0..5] OF Vec3;
	lstJntPos: ARRAY[0..5] OF Vec3;
	jntFce : ARRAY[0..5] OF Vec3;
	tipFce : ARRAY[0..5] OF Vec3;//2G
	tipFce2B : ARRAY[0..5] OF Vec3;
	tipFce2H : ARRAY[0..5] OF Vec3;
	
	stepL : LREAL;//直线距离
	stepDir : LREAL;
    stepYaw : LREAL;//dyaw
	deltaT : LREAL;
	swingID : ARRAY[0..2] OF DINT;
	stanceID : ARRAY[0..2] OF DINT;
	isAllContact : BOOL;
	allContactTime: LREAL;
	
	lstRollErr: LREAL:=0;
	lstPitchErr: LREAL:=0;
	sumRollErr: LREAL:=0;
	sumPitchErr: LREAL:=0;
	kp:LREAL:=1000;
	ki:LREAL:=3000;//对效果影响较大，kp的1-4倍效果差不多
	kd:LREAL:=100;//和0差别不明显
	kRatio:LREAL:=2;//pitch方向增益要给大点，通过该参数控制
	wrench: Vec3;
	fceStance: Vec3;
	readyToRelease: BOOL;
END_VAR

METHOD Arc2Line : BOOL
//步长通过弧长定义，但计算需要直线距离
VAR_INPUT
	arcLen: LREAL;
	angle: LREAL;
END_VAR
VAR_OUTPUT
	lineLen: LREAL;
END_VAR
VAR
	radius: LREAL;
END_VAR
IF ABS(angle) < 0.001 THEN
	lineLen := arcLen;
ELSE
	lineLen := arcLen * SIN(angle/2) / (angle/2);
END_IF
END_METHOD

METHOD BodyPlanning : BOOL
VAR_INPUT
	count: DINT;
END_VAR
VAR
	HmItp: HermitInterpolation;
	i: INT;
	t: LREAL;
	decRatio: LREAL;
	delta: ARRAY[0..2] OF LREAL;
END_VAR
//xyz在bodyTrgt坐标系内规划后转换至地面坐标系
//xy据不同触地时间动态调整
t := count*deltaT;
decRatio := 0.2;
delta[0] := decRatio/2*stepL*COS(stepDir)*COS(decRatio/2*stepYaw/2)
           -decRatio/2*stepL*SIN(stepDir)*SIN(decRatio/2*stepYaw/2);
delta[1] := decRatio/2*stepL*COS(stepDir)*SIN(decRatio/2*stepYaw/2)
           +decRatio/2*stepL*SIN(stepDir)*COS(decRatio/2*stepYaw/2);
IF t <= allContactTime + period THEN
	FOR i:=0 TO 1 DO
		HmItp(t0:=allContactTime,T:=period,
			  y0:=bodyPosInit2T.data[i],y1:=0,
			  v0:=bodyVelInit2T.data[i],v1:=bodyVelTrgt2T.data[i],
			  tNow:=t,
			  y=>bodyPos2T.data[i],v=>bodyVel2T.data[i]);
	END_FOR
ELSIF t <= allContactTime + period + decRatio * period THEN
	FOR i:=0 TO 1 DO
		HmItp(t0:=allContactTime+period,T:=decRatio*period,
			  y0:=0,y1:=delta[i],
			  v0:=bodyVelTrgt2T.data[i],v1:=0,
			  tNow:=t,
			  y=>bodyPos2T.data[i],v=>bodyVel2T.data[i]);
	END_FOR
ELSE
	FOR i:=0 TO 1 DO
		bodyPos2T.data[i] := delta[i];
		bodyVel2T.data[i] := 0;
	END_FOR
END_IF
//z前1/2周期完成调整后不变
IF t <= allContactTime + period/2 THEN
	HmItp(t0:=allContactTime,T:=period/2,
		  y0:=bodyPosInit2T.data[2],y1:=0,
		  v0:=0,v1:=0,
		  tNow:=t,
		  y=>bodyPos2T.data[2],v=>bodyVel2T.data[2]);
ELSE
	bodyPos2T.data[2] := 0;
	bodyVel2T.data[2] := 0;
END_IF
//转换至地面坐标系
bodyPos := VecAdd(MatMulVec(bodyPmxTrgt,bodyPos2T),bodyPosTrgt);
bodyVel := MatMulVec(bodyPmxTrgt,bodyVel2T);

//rpy在地面坐标系内规划
//roll,pitch在1/2周期内完成调整后不变
IF t <= allContactTime + period/2 THEN
	FOR i:=0 TO 1 DO
		HmItp(t0:=allContactTime,T:=period/2,
			  y0:=bodyRPYInit.data[i],y1:=bodyRPYTrgt.data[i],
			  v0:=0,v1:=0,
			  tNow:=t,
			  y=>bodyRPY.data[i]);
	END_FOR
ELSE
	FOR i:=0 TO 1 DO
		bodyRPY.data[i] := bodyRPYTrgt.data[i];
	END_FOR
END_IF
//yaw据不同触地时间动态调整
delta[2] := decRatio/2*stepYaw;
IF t <= allContactTime + period THEN
	HmItp(t0:=allContactTime,T:=period,
		  y0:=bodyRPYInit.data[2],y1:=bodyRPYTrgt.data[2],
		  v0:=bodyOmgInit,v1:=bodyOmgTrgt,
		  tNow:=t,
		  y=>bodyRPY.data[2],v=>bodyOmg);
ELSIF t <= allContactTime + period + decRatio * period THEN
	HmItp(t0:=allContactTime+period,T:=decRatio*period,
		  y0:=bodyRPYTrgt.data[2],y1:=bodyRPYTrgt.data[2]+delta[2],
		  v0:=bodyOmgTrgt,v1:=0,
		  tNow:=t,
		  y=>bodyRPY.data[2],v=>bodyOmg);
ELSE
	bodyRPY.data[2] := bodyRPYTrgt.data[2]+delta[2];
	bodyOmg := 0;
END_IF
objRotMtx(yaw:=bodyRPY.data[2],pitch:=bodyRPY.data[1],roll:=bodyRPY.data[0],rm=>bodyPmx);
END_METHOD

METHOD CalcAddfce : BOOL
VAR_INPUT
	count: UDINT;
END_VAR
VAR_OUTPUT
END_VAR
VAR
	maxAddFce:LREAL;
	maxFceStance:LREAL;
	fmatStance: Mat3;
	//fceStance: Vec3;
	maxFceSwing:LREAL;
	fmatSwing: Mat3;
	fceSwing: Vec3;
	
	rollErr: LREAL;
	pitchErr: LREAL;
	difRollErr: LREAL;
	difPitchErr: LREAL;
	//wrench: Vec3;
	
	tipFceTmp: ARRAY[0..5] OF Vec3;
	ratio: ARRAY[0..5] OF LREAL;
	i: INT;
	j: INT;
	step: LREAL;
	t: LREAL;
END_VAR
maxAddFce:=800;
step:=4;
//IF isAllContact=TRUE THEN
//	sumRollErr:=0;
//	sumPitchErr:=0;
//END_IF

rollErr:=bodyRPY.data[0]-gvl.rpy_model[0];
pitchErr:=bodyRPY.data[1]-gvl.rpy_model[1];
IF ABS(rollErr) < 0.002 THEN
	rollErr:=0;
END_IF
IF ABS(pitchErr) < 0.002 THEN
	pitchERr:=0;
END_IF
sumRollErr:=sumRollErr+rollErr*deltaT;
difRollErr:=(rollErr-lstRollErr)/deltaT;
sumPitchErr:=sumPitchErr+pitchErr*deltaT;
difPitchErr:=(pitchErr-lstPitchErr)/deltaT;
lstRollErr:=rollErr;
lstPitchErr:=pitchErr;

wrench.data[0]:=kp*rollErr+ki*sumRollErr+kd*difRollErr;
wrench.data[1]:=kRatio*(kp*pitchErr+ki*sumPitchErr+kd*difPitchErr);
wrench.data[2]:=600;//gravity

//stance leg
fmatStance:=setMat3(tipPos[stanceID[0]].data[1]-bodyPos.data[1],tipPos[stanceID[1]].data[1]-bodyPos.data[1],tipPos[stanceID[2]].data[1]-bodyPos.data[1],
              -tipPos[stanceID[0]].data[0]+bodyPos.data[0],-tipPos[stanceID[1]].data[0]+bodyPos.data[0],-tipPos[stanceID[2]].data[0]+bodyPos.data[0],
              1,1,1);
fceStance:=MatMulVec(inv3(fmatStance),wrench);
maxFceStance:=MAX(ABS(fceStance.data[0]),ABS(fceStance.data[1]),ABS(fceStance.data[2]));
IF maxFceStance>maxAddFce THEN
	FOR i:=0 TO 2 DO
		tipFceTmp[stanceID[i]]:=SetVec3(0,0,-fceStance.data[i]/maxFceStance*maxAddFce);
	END_FOR
ELSE	
	FOR i:=0 TO 2 DO
		tipFceTmp[stanceID[i]]:=SetVec3(0,0,-fceStance.data[i]);
	END_FOR
END_IF
//swing leg
(*fmatSwing:=setMat3(tipPos[swingID[0]].data[1]-bodyPos.data[1],tipPos[swingID[1]].data[1]-bodyPos.data[1],tipPos2B[swingID[2]].data[1]-bodyPos.data[1],
              -tipPos2B[swingID[0]].data[0]+bodyPos.data[0],-tipPos2B[swingID[1]].data[0]+bodyPos.data[0],-tipPos2B[swingID[2]].data[0]+bodyPos.data[0],
              1,1,1);
fceSwing:=MatMulVec(inv3(fmatSwing),wrench);
maxFceSwing:=MAX(ABS(fceSwing.data[0]),ABS(fceSwing.data[1]),ABS(fceSwing.data[2]));
IF maxFceSwing>maxAddFce THEN
	FOR i:=0 TO 2 DO
		tipFceTmp[swingID[i]]:=SetVec3(0,0,-fceSwing.data[i]/maxFceSwing*maxAddFce);
	END_FOR
ELSE	
	FOR i:=0 TO 2 DO
		tipFceTmp[swingID[i]]:=SetVec3(0,0,-fceSwing.data[i]);
	END_FOR
END_IF*)

//方法1,空中给摆动腿加力，感觉只会导致更提前触地，并不能改善倾斜
(*
t := count*deltaT;
IF ABS(t-allContactTime)<deltaT THEN
	FOR i:=0 TO 5 DO
		ratio[i]:=1;
	END_FOR
END_IF
FOR i:=0 TO 2 DO
	IF t-allContactTime<period/2 THEN
		ratio[swingID[i]]:=ratio[swingID[i]]*0.99;//1-0
	ELSE
		ratio[swingID[i]]:=ratio[swingID[i]]/0.99;//0-1
	END_IF
	IF ratio[swingID[i]]>1 THEN//限制在0.01~1
		ratio[swingID[i]]:=1;
	END_IF
	IF ratio[swingID[i]]<0.01 THEN
		ratio[swingID[i]]:=0.01;
	END_IF
	tipFce[stanceID[i]].data[2]:=ratio[stanceID[i]]*tipFceTmp[stanceID[i]].data[2];
	tipFce[swingID[i]].data[2]:=ratio[swingID[i]]*tipFceTmp[swingID[i]].data[2];
END_FOR*)

//方法2
FOR i:=0 TO 2 DO
	IF tipFceTmp[stanceID[i]].data[2]-tipFce[stanceID[i]].data[2]>step THEN
		tipFce[stanceID[i]].data[2]:=tipFce[stanceID[i]].data[2]+step;
	ELSIF tipFceTmp[stanceID[i]].data[2]-tipFce[stanceID[i]].data[2]<-step THEN
		tipFce[stanceID[i]].data[2]:=tipFce[stanceID[i]].data[2]-step;
	ELSE
		tipFce[stanceID[i]].data[2]:=tipFce[stanceID[i]].data[2];
	END_IF
END_FOR

FOR i:=0 TO 2 DO
	tipFce[swingID[i]]:=SetVec3(0,0,tipFce[swingID[i]].data[2]*0.995);
END_FOR

FOR i:=0 TO 5 DO
	tipFce2B[i] := MatMulVec(MatTranspose(bodyPmx),     tipFce[i]);
	tipFce2H[i] := MatMulVec(MatTranspose(hipPmx2B[i]), tipFce2B[i]);
	gvl.legCtrl[i].DesireDriveForce(fTipDes:=tipFce2H[i].data,motorAng:=jntPos[i].data,
                                    legIndex:=i,fDrvDes=>jntFce[i].data);
END_FOR
END_METHOD

METHOD CalcSlope : BOOL
VAR_INPUT
	yaw: LREAL;
END_VAR
VAR_OUTPUT
	roll: LREAL;
	pitch: LREAL;
	deltaH: LREAL;//身体需调整的高度
	tipDelta: Vec3;//足尖需调整的距离
END_VAR
VAR
	i: INT;
	bodyActualPmx: Mat3;
	tipActualPos2H: Vec3;
	tipActualPos2B: Vec3;
	tipActPos: ARRAY[0..5] OF Vec3;
	va1 : Vec3;
	vb1 : Vec3;
	vz1 : Vec3;
	va2 : Vec3;
	vb2 : Vec3;
	vz2 : Vec3;
	vz  : Vec3;
	avgTipZ: LREAL;
	actualH: LREAL;
END_VAR
objRotMtx(yaw:=0,pitch:=GVL.rpy_model[1],roll:=GVL.rpy_model[0],
		  rm=>bodyActualPmx);
FOR i:=0 TO 5 DO
	tipActualPos2H:=SetVec3(GVL.tipActualPos[i,0],GVL.tipActualPos[i,1],GVL.tipActualPos[i,2]);
	tipActualPos2B:=VecAdd(MatMulVec(hipPmx2B[i],tipActualPos2H),hipPos2B[i]);
	tipActPos[i]:=VecAdd(MatMulVec(bodyActualPmx,tipActualPos2B),bodyPos);
END_FOR
//用tipActPos替代tipPos看效果
va1 := SetVec3(tipActPos[stanceID[0]].data[0]-tipActPos[stanceID[1]].data[0],
	          tipActPos[stanceID[0]].data[1]-tipActPos[stanceID[1]].data[1],
			  tipActPos[stanceID[0]].data[2]-tipActPos[stanceID[1]].data[2]);
vb1 := SetVec3(tipActPos[stanceID[0]].data[0]-tipActPos[stanceID[2]].data[0],
	          tipActPos[stanceID[0]].data[1]-tipActPos[stanceID[2]].data[1],
			  tipActPos[stanceID[0]].data[2]-tipActPos[stanceID[2]].data[2]);
vz1 := VecNormalize(VecCross(va1,vb1));
IF vz1.data[2]<0 THEN//保证vz朝上
	vz1 := VecNeg(vz1);
END_IF
va2 := SetVec3(tipActPos[swingID[0]].data[0]-tipActPos[swingID[1]].data[0],
	          tipActPos[swingID[0]].data[1]-tipActPos[swingID[1]].data[1],
			  tipActPos[swingID[0]].data[2]-tipActPos[swingID[1]].data[2]);
vb2 := SetVec3(tipActPos[swingID[0]].data[0]-tipActPos[swingID[2]].data[0],
	          tipActPos[swingID[0]].data[1]-tipActPos[swingID[2]].data[1],
			  tipActPos[swingID[0]].data[2]-tipActPos[swingID[2]].data[2]);
vz2 := VecNormalize(VecCross(va2,vb2));
IF vz2.data[2]<0 THEN//保证vz朝上
	vz2 := VecNeg(vz2);
END_IF

vz := VecNormalize(VecAdd(vz1,vz2));

//trgtPmxB2G*z=vz,求出trgtPmx对应的roll和pitch
roll  := ASIN(  vz.data[0]*SIN(yaw)-vz.data[1]*COS(yaw) );
pitch := ATAN( (vz.data[0]*COS(yaw)+vz.data[1]*SIN(yaw)) / vz.data[2] );

//地面坐标系
//avgTipZ := (tipPos[stanceID[0]].data[2]+tipPos[stanceID[1]].data[2]+tipPos[stanceID[2]].data[2])/3;
//actualH := bodyPos[2]-avgTipZ;//地面坐标系内身体实际高度
//deltaH := bodyRefH / vz.data[2] - actualH;
//身体坐标系
avgTipZ := (tipActPos[stanceID[0]].data[2]+tipActPos[stanceID[1]].data[2]+tipActPos[stanceID[2]].data[2]
           +tipActPos[swingID[0]].data[2]+tipActPos[swingID[1]].data[2]+tipActPos[swingID[2]].data[2])/6;
actualH := bodyPos.data[2]-avgTipZ;//地面坐标系内身体实际高度
deltaH := bodyRefH - actualH*vz.data[2];

//地面坐标系
//垂直坡面方向高度向量，减去竖直方向高度向量
tipDelta := VecAdd( VecMulNum(vz,bodyRefH),SetVec3(0,0,-bodyRefH/vz.data[2]) );
END_METHOD

METHOD DoPlanning : BOOL
VAR_INPUT
	count: UDINT;
END_VAR
VAR
	i,j : INT;	
	tmpID: ARRAY [0..2] OF DINT;
	
	(*init var*)
	(*bodyWid  : LREAL := 0.306;
	bodyLen  : LREAL := 0.712;
	bodyLen2 : LREAL := 0.250;
	bodyAng  : LREAL := pi/4;
	tipYsum : LREAL;*)
END_VAR
IF count = 0 THEN
	Initialize();
	(*
	hipPos2B[0] := SetVec3( -bodyLen2/2,  bodyWid/2, 0);
	hipPos2B[1] := SetVec3(  bodyLen2/2,  bodyWid/2, 0);
	hipPos2B[2] := SetVec3(   bodyLen/2,          0, 0);
	hipPos2B[3] := SetVec3(  bodyLen2/2, -bodyWid/2, 0);
	hipPos2B[4] := SetVec3( -bodyLen2/2, -bodyWid/2, 0);
	hipPos2B[5] := SetVec3(  -bodyLen/2,          0, 0);
	
	objRotMtx(yaw:=-bodyAng   , pitch:=0, roll:=pi/2, rm=>hipPmx2B[0]);
	objRotMtx(yaw:= bodyAng+pi, pitch:=0, roll:=pi/2, rm=>hipPmx2B[1]);
	objRotMtx(yaw:=         pi, pitch:=0, roll:=pi/2, rm=>hipPmx2B[2]);
	objRotMtx(yaw:=-bodyAng+pi, pitch:=0, roll:=pi/2, rm=>hipPmx2B[3]);
	objRotMtx(yaw:= bodyAng   , pitch:=0, roll:=pi/2, rm=>hipPmx2B[4]);
	objRotMtx(yaw:= 0         , pitch:=0, roll:=pi/2, rm=>hipPmx2B[5]);
	
	//获取初始关节位置
	FOR i:=0 TO 5 DO
		FOR j:=0 TO 2 DO
			jntPosInit[i].data[j] := gvl.jntLastRefPos[i,j];
		END_FOR
	END_FOR
	
	//获取初始身体和足尖位置
	tipYSum := 0;
	FOR i:=0 TO 5 DO
		gvl.legCtrl[i].ForwardKinetics(motorAngles := jntPosInit[i].data,legIndex := i,tipPosition => tipPosInit2H[i].data);
		tipYSum := tipYSum + tipPosInit2H[i].data[1];
	END_FOR
	bodyRefH := -tipYSum/6.0;//positive
	bodyPosInit := SetVec3(0, 0, 0);
	bodyRPYInit := SetVec3(gvl.rpy_model[0],gvl.rpy_model[1],0);
	objRotMtx(yaw:=0,pitch:=gvl.rpy_model[1],roll:=gvl.rpy_model[0],rm=>bodyPmxInit);
	
	FOR i:=0 TO 5 DO
		tipPosInit2B[i]:=VecAdd(MatMulVec(hipPmx2B[i],tipPosInit2H[i]),hipPos2B[i]);
		tipPosInit[i]:=VecAdd(MatMulVec(bodyPmxInit,tipPosInit2B[i]),bodyPosInit);
	END_FOR
	
	//初始化规划变量
	bodyPos := bodyPosInit;
	bodyRPY := bodyRPYInit;
	tipPos := tipPosInit;
	tipPos2H := tipPosInit2H;
	
	FOR i := 0 TO 5 DO
		FOR j := 0 TO 2 DO
			jointPosTarget[i, j] := jntPosInit[i].data[j];
			jointVelTarget[i, j] := 0;
			jointFceTarget[i, j] := 0;
			lstJntPos[i].data[j] := jntPosInit[i].data[j];
		END_FOR
	END_FOR*)
	
	deltaT := 1.0 / gvl.sampleRate;
	isAllContact := TRUE;
	allContactTime := 0;
	isFinished := FALSE;
	isLastStep := FALSE;
	FOR i:=0 TO 2 DO
		swingID[i] := 2*i;
		stanceID[i] := 2*i+1;
	END_FOR
	bodyVel := SetVec3(0,0,0);
	bodyOmg := 0;
END_IF

//WatchDog(count);
IF isAllContact = TRUE THEN
	//状态更新
	isAllContact := FALSE;
	tmpID := swingID;
	swingID := stanceID;
	stanceID := tmpID;
	
	//处理第一步、最后一步的不同步长、速度
	IF count = 0 THEN//first step
		stepL := SQRT(cmdL*cmdL+cmdLa*cmdLa)/2;
		stepDir := Atan2(cmdLa,cmdL);
		stepYaw := cmdYaw/180*pi / 2;
		bodyVelTrgt2T := SetVec3(cmdL/period,cmdLa/period,0);
		bodyOmgTrgt := cmdYaw/180*pi / period;
	ELSIF isLastStep = TRUE THEN//last step
		stepL := SQRT(cmdL*cmdL+cmdLa*cmdLa)/2;
		stepDir := Atan2(cmdLa,cmdL);
		stepYaw := cmdYaw/180*pi / 2;
		bodyVelTrgt2T := SetVec3(0,0,0);
		bodyOmgTrgt := 0;
	ELSE
		stepL := SQRT(cmdL*cmdL+cmdLa*cmdLa);
		stepDir := Atan2(cmdLa,cmdL);
		stepYaw := cmdYaw/180*pi;
		bodyVelTrgt2T := SetVec3(cmdL/period,cmdLa/period,0);
		bodyOmgTrgt := cmdYaw/180*pi / period;
	END_IF
	
	UpdateInitAndTrgt();
END_IF

IF readyToRelease=FALSE THEN
	BodyPlanning(count);
	FOR i:=0 TO 2 DO
		SwingPlanning(count,swingID[i]);
		//StancePlanning-->do nothing;
	END_FOR
END_IF
//else do no planning

IF isContact(count,swingID[0]) = TRUE AND VecNorm(tipVel[swingID[0]]) < 1E-3 AND
   isContact(count,swingID[1]) = TRUE AND VecNorm(tipVel[swingID[1]]) < 1E-3 AND
   isContact(count,swingID[2]) = TRUE AND VecNorm(tipVel[swingID[2]]) < 1E-3 THEN
   isAllContact := TRUE;
   allContactTime := count*deltaT;
END_IF

//计算hip坐标系内足尖位置-->关节位置速度
IF readyToRelease=FALSE THEN
	FOR i:=0 TO 5 DO
		tipPos2B[i] := MatMulVec(MatTranspose(bodyPmx),    VecAdd(tipPos[i],  VecNeg(bodyPos)));
		tipPos2H[i] := MatMulVec(MatTranspose(hipPmx2B[i]),VecAdd(tipPos2B[i],VecNeg(hipPos2B[i])));
		gvl.legCtrl[i].InverseKinetics(tipPosition := tipPos2H[i].data, refPosLast:=lstJntPos[i].data,legIndex:=i,
									   motorAngles => jntPos[i].data);
		jntVel[i] := VecAdd(jntPos[i],VecNeg(lstJntPos[i]));
		lstJntPos[i] := jntPos[i];
	END_FOR
	CalcAddfce(count);
END_IF
//else do no planning

// link to physical outputs
FOR i := 0 TO 5 DO
	FOR j := 0 TO 2 DO
		jointPosTarget[i, j] := jntPos[i].data[j];
		jointVelTarget[i, j] := jntVel[i].data[j];
		IF readyToRelease=FALSE THEN
			jointFceTarget[i, j] := jntFce[i].data[j];
		END_IF
	END_FOR
END_FOR

IF isLastStep=TRUE AND isAllContact=TRUE THEN
	readyToRelease := TRUE;
	isLastStep := FALSE;
END_IF
IF readyToRelease=TRUE THEN//use 50 count to release
	FOR i := 0 TO 5 DO
		FOR j := 0 TO 2 DO
			jointFceTarget[i, j] := jointFceTarget[i, j]-0.02*jntFce[i].data[j];
		END_FOR
	END_FOR
	IF count*deltaT-allContactTime>=50*deltaT THEN
		isFinished := TRUE;
	END_IF
END_IF
END_METHOD

METHOD Initialize : BOOL
VAR_INPUT
END_VAR

VAR
	i,j : UINT;
	tipYsum : LREAL;
	offset0 : Vec3;
	offset5 : Vec3;
END_VAR
hipPmx2B[0]:=SetMat3(1,0,0,0,0,-1,0,1,0);
hipPmx2B[1]:=SetMat3(-1,0,0,0,0,1,0,1,0);
hipPmx2B[2]:=SetMat3(-1,0,0,0,0,1,0,1,0);
hipPmx2B[3]:=SetMat3(-1,0,0,0,0,1,0,1,0);
hipPmx2B[4]:=SetMat3(-1,0,0,0,0,1,0,1,0);
hipPmx2B[5]:=SetMat3(1,0,0,0,0,-1,0,1,0);

hipPos2B[0] := SetVec3(-0.369, -0.125, 0);
hipPos2B[1] := SetVec3(     0,  -0.28, 0);
hipPos2B[2] := SetVec3(  0.36, -0.125, 0);
hipPos2B[3] := SetVec3(  0.36,  0.125, 0);
hipPos2B[4] := SetVec3(     0,   0.28, 0);
hipPos2B[5] := SetVec3(-0.369,  0.125, 0);

//获取初始关节位置
FOR i:=0 TO 5 DO
	FOR j:=0 TO 2 DO
		jntPosInit[i].data[j] := gvl.jntLastRefPos[i,j];
	END_FOR
END_FOR

//获取初始身体和足尖位置
tipYSum := 0;
FOR i:=0 TO 5 DO
	gvl.legCtrl[i].ForwardKinetics(motorAngles := jntPosInit[i].data,legIndex:=i,tipPosition => tipPosInit2H[i].data);
	tipYSum := tipYSum + tipPosInit2H[i].data[1];
END_FOR
bodyRefH := -tipYSum/6.0;//positive
bodyPosInit := SetVec3(0, 0, 0);
bodyRPYInit := SetVec3(gvl.rpy_model[0],gvl.rpy_model[1],0);
objRotMtx(yaw:=0,pitch:=gvl.rpy_model[1],roll:=gvl.rpy_model[0],rm=>bodyPmxInit);

FOR i:=0 TO 5 DO
	tipPosInit2B[i]:=VecAdd(MatMulVec(hipPmx2B[i],tipPosInit2H[i]),hipPos2B[i]);
	tipPosTrgtBase[i]:=tipPosInit2B[i];
	IF i=0 THEN
		tipPosTrgtBase[i].data[1]:=tipPosTrgtBase[i].data[1]-0.03;
	ELSIF i=5 THEN
		tipPosTrgtBase[i].data[1]:=tipPosTrgtBase[i].data[1]+0.03;
	END_IF
	tipPosInit[i]:=VecAdd(MatMulVec(bodyPmxInit,tipPosInit2B[i]),bodyPosInit);
END_FOR

//初始化规划变量
bodyPos := bodyPosInit;
bodyRPY := bodyRPYInit;
tipPos := tipPosInit;
tipPos2H := tipPosInit2H;

FOR i := 0 TO 5 DO
	FOR j := 0 TO 2 DO
		jointPosTarget[i, j] := jntPosInit[i].data[j];
		jointVelTarget[i, j] := 0;
		jointFceTarget[i, j] := 0;
		lstJntPos[i].data[j] := jntPosInit[i].data[j];
	END_FOR
	tipFce[i]:=SetVec3(0,0,0);
END_FOR

lstRollErr:=0;
lstPitchErr:=0;
sumRollErr:=0;
sumPitchErr:=0;
readyToRelease:=FALSE;
END_METHOD

METHOD isContact : BOOL
VAR_INPUT
	count: DINT;
	legID: DINT;
END_VAR
VAR
	fceLimit : LREAL;
END_VAR
IF legID = 0 OR legID = 5 THEN
	fceLimit := 80;
ELSE
	fceLimit := 60;
END_IF

//IF count*deltaT > allContactTime+period THEN//离线测试
IF count*deltaT > allContactTime+period/4 AND  gvl.tipActualFce[legID,1] > fceLimit THEN
	isContact := TRUE;
ELSE
	isContact := FALSE;
END_IF
END_METHOD

METHOD SwingPlanning : BOOL
VAR_INPUT
	count: DINT;
	legID: DINT;
END_VAR
VAR
	i: INT;
	t: LREAL;
	tp: ARRAY[0..4] OF LREAL;
	xp: ARRAY[0..4] OF LREAL;
	yp: ARRAY[0..4] OF LREAL;
	zp: ARRAY[0..4] OF LREAL;
	landVel: LREAL;
	decTime: LREAL;
	acc: LREAL;
	objSpline: CubicSpline;
END_VAR
//generate 5 waypoints
tp[0] := allContactTime;
tp[1] := tp[0] + period / 6;
tp[2] := tp[1] + period / 6;
tp[3] := tp[2] + period / 3;
tp[4] := tp[3] + period / 3;

xp[0] := tipPosInit[legID].data[0];
yp[0] := tipPosInit[legID].data[1];
zp[0] := tipPosInit[legID].data[2];

xp[4] := tipPosTrgt[legID].data[0];
yp[4] := tipPosTrgt[legID].data[1];
zp[4] := tipPosTrgt[legID].data[2];

xp[1] := xp[0] - swingDir * cmdH/2;//0 or 1
yp[1] := yp[0];
zp[1] := zp[0] + cmdH/2;

xp[3] := xp[4];
yp[3] := yp[4];
zp[3] := zp[4] + cmdH/2;

xp[2] := (xp[0]+xp[4])/2;
yp[2] := (yp[0]+yp[4])/2;
zp[2] := (zp[0]+zp[4])/2 + cmdH;

